(*Pump States*)
IF (iq_stPtm.i_xFault) THEN
        iq_stPtm.eState := pumpFAULT;
        iq_stPtm.xRunSW:=FALSE;
        q_RunDO:=FALSE;
ELSIF (iq_stPtm.q_RunDO) AND (iq_stPtm.i_xAtSpd) THEN
        iq_stPtm.eState := pumpRUNNING;
ELSIF (iq_stPtm.q_RunDO) AND NOT (iq_stPtm.i_xAtSpd) THEN
        iq_stPtm.eState := pumpSTARTING;
ELSIF NOT (iq_stPtm.q_RunDO) THEN
        iq_stPtm.eState := pumpSTOPPED;
ELSE
    iq_stPtm.eState := pumpFAULT;
END_IF;


(*I/O soft mapping*)
ACT_IO();
// Log States and triggers
This^.ACT_Logger();
(*Load or save the persistent variables*)
ACT_Persistent();

ACTION ACT_IO:
(*Inputs*)
iq_stPtm.i_xAtSpd := i_xAtSpd;
iq_stPtm.i_xNCError := i_xFaultNC;
iq_stPtm.i_xFault := NOT i_xFaultNC;



(*Outputs*)
iq_stPtm.q_RunDO := q_RunDO;
END_ACTION

ACTION ACT_Logger:
//STATE Logger
// ILK logger
IF NOT i_xExtIlkOK AND ePrevState = pumpRUNNING THEN
         fbLogger(sMsg:='Lost external interlock while pump was running.', eSevr:=TcEventSeverity.Critical);
END_IF


IF ePrevState <> iq_stPTM.eState THEN
      CASE iq_stPTM.eState OF
        pumpFAULT:
            fbLogger(sMsg:='Pump Fault.', eSevr:=TcEventSeverity.Critical);
          pumpSTOPPED:
            fbLogger(sMsg:='Pump stopped.', eSevr:=TcEventSeverity.Critical);
        pumpSTARTING:
            fbLogger(sMsg:='Pump starting.', eSevr:=TcEventSeverity.Info);
        pumpRUNNING:
            fbLogger(sMsg:='Pump running.', eSevr:=TcEventSeverity.Info);
      END_CASE
      ePrevState := iq_stPTM.eState;
  END_IF

// Log Action
tAction(CLK:=  iq_stPTM.q_RunDO);
IF tAction.Q THEN fbLogger(sMsg:='Pump commanded to start', eSevr:=TcEventSeverity.Info); END_IF


// Log FAULT
tFault(CLK:= NOT iq_stPTM.i_xFault);
IF tFault.Q THEN fbLogger(sMsg:='Pump Lost Alarm OK bit', eSevr:=TcEventSeverity.Critical); END_IF
END_ACTION

ACTION ACT_Persistent:
(*On first PLC pass, load the persistent value into the structrue variable*)
IF (SUPER^.bRestorePersistentData) THEN
    SUPER^.bRestorePersistentData	:= FALSE;
    IF (rBackingPressureSP <> 0) THEN
        iq_stPTM.rBackingPressureSP := rBackingPressureSP;
    END_IF;
    IF (rInletPressureSP <> 0) THEN
        iq_stPTM.rInletPressureSP := rInletPressureSP;
    END_IF;
END_IF
(*Check if a new value has been written in the structure variable copy it to the persistent variable*)
IF NOT (iq_stPTM.rBackingPressureSP = rBackingPressureSP) THEN
    rBackingPressureSP:= iq_stPTM.rBackingPressureSP;
END_IF;

IF NOT (iq_stPTM.rInletPressureSP = rInletPressureSP) THEN
    rInletPressureSP := iq_stPTM.rInletPressureSP;
END_IF;
END_ACTION

METHOD PUBLIC M_Run : BOOL
VAR_INPUT
    run:bool; // set to true to run, false to stop;
END_VAR

this^.iq_stPtm.xRunSW := run;
END_METHOD

METHOD PUBLIC M_Serial_IO : BOOL
VAR_INPUT
    i_st_TD20_RBK			: ST_TD20Status;
END_VAR

(* This function block is used to map the IO points from the Oerlikon structures
to the generic turbo structures *)

(* Readbacks *)
iq_stPTM.i_xAccel := i_st_TD20_RBK.wStatusWord.4;
iq_stPTM.i_xDecel := i_st_TD20_RBK.wStatusWord.5;
//iq_stPTM.i_xAtSpd := i_st_TD20_RBK.wStatusWord.10;
iq_stPTM.i_xRemote := i_st_TD20_RBK.wStatusWord.15; (* Remote control enabled *)
iq_stPTM.i_diCurSpd := WORD_TO_DINT(i_st_TD20_RBK.wFrequency_P3);
iq_stPTM.i_rCurrentMon := WORD_TO_INT(i_st_TD20_RBK.wMotorCurrent_P5)*0.1; (*Current in units 0.1 A, TD20 manual page 23*)
iq_stPTM.i_diPwr := LREAL_TO_DINT(WORD_TO_DINT(i_st_TD20_RBK.wMotorCurrent_P5 * i_st_TD20_RBK.wVoltage_P4)*0.01); (*Current in units 0.1 A and voltage in units 0.1V, TD20 manual page 23*)
iq_stPTM.i_diElecTemp := WORD_TO_DINT(i_st_TD20_RBK.wConverterTemp_P11);
iq_stPTM.i_rTempMon := WORD_TO_INT(i_st_TD20_RBK.wPumpTemp_P127);

(* Faults and warnings *)
//iq_stPTM.i_xFault := i_st_TD20_RBK.wStatusWord.3;
iq_stPTM.i_xTempFault := i_st_TD20_RBK.wStatusWord.7; (* specified as a temperature warning but it could be a fault *)
iq_stPTM.i_xWarn := i_st_TD20_RBK.wStatusWord.14; (* warning summary bit *)
END_METHOD

METHOD PUBLIC M_SetBackingSP
VAR_INPUT
    i_fBackingPressureSP : REAL;
END_VAR
iq_stPtm.rBackingPressureSP := i_fBackingPressureSP;
END_METHOD

METHOD PUBLIC M_SetForelineSP
VAR_INPUT
    i_fForelinePressureSP : REAL;
END_VAR
iq_stPtm.rForelineSP := i_fForelinePressureSP;
END_METHOD

END_FUNCTION_BLOCK

// ---- POUs/Functions/Pumps/FB_PTM_TwisTorr.TcPOU
(* This function block does basic controls FOR the Agilent TwisTorr 304 FS with on board Controller.
 Turns off pump in the event of errors/ warnings. Provides interlocking interface.*)
FUNCTION_BLOCK FB_PTM_TwisTorr EXTENDS FB_Pump
VAR_INPUT
    i_xExtILKOk : BOOL; // Connect to external interlock logic, TRUE if not used.
END_VAR
VAR_OUTPUT
    {attribute 'pytmc' := ' pv: '}
    iq_stPtm	:	ST_PTM;
END_VAR
VAR
    xRunOk	:	BOOL;
    (*IO*)
    i_xAtSpd AT%I*: BOOL; // Normaml operation when true
    i_xFault AT%I*: BOOL; // Error // this open collector output signal is ON when a system fault condition is detected
    q_RunDO AT%Q*: BOOL; // Start/Stop
END_VAR


(* Interlock Sum *)
iq_stPtm.xExtRunOk:= i_xExtILKOk;
xRunOk := iq_stPtm.xExtRunOk AND NOT iq_stPtm.i_xFault;

(* Basic pump supervisory section *)
IF xRunOk THEN
    iq_stPtm.q_RunDO := iq_stPTM.xRunSW;
ELSE
    iq_stPtm.xRunSW:=FALSE;
    iq_stPtm.q_RunDO:=FALSE;
END_IF

(*Pump STATE*)
IF iq_stPtm.i_xFault THEN
    iq_stPtm.eState := pumpFAULT;
ELSIF NOT iq_stPtm.q_RunDO AND NOT iq_stPTM.i_xFault THEN
    iq_stPtm.eState := pumpSTOPPED;
ELSIF NOT iq_stPtm.i_xAtSpd  AND iq_stPtm.q_RunDO THEN
    iq_stPtm.eState := pumpSTARTING;
ELSIF iq_stPtm.i_xAtSpd AND iq_stPtm.q_RunDO THEN
    iq_stPtm.eState := pumpRUNNING;
ELSE
    iq_stPtm.eState := pumpFAULT;
END_IF

(*I/O soft mapping*)
ACT_IO();
(*Log States and triggers*)
ACT_Logger();
(*Load or save the persistent variables*)
ACT_Persistent();

ACTION ACT_IO:
(*Inputs*)
iq_stPtm.i_xAtSpd := i_xAtSpd;
iq_stPtm.i_xFault := i_xFault;


(*Outputs*)
q_RunDO := iq_stPtm.q_RunDO;
END_ACTION

ACTION ACT_Logger:
//STATE Logger
// ILK logger
IF NOT i_xExtIlkOK AND ePrevState = pumpRUNNING THEN
         fbLogger(sMsg:='Lost external interlock while pump was running.', eSevr:=TcEventSeverity.Critical);
END_IF


IF ePrevState <> iq_stPTM.eState THEN
      CASE iq_stPTM.eState OF
        pumpFAULT:
            fbLogger(sMsg:='Pump Fault.', eSevr:=TcEventSeverity.Critical);
          pumpSTOPPED:
            fbLogger(sMsg:='Pump stopped.', eSevr:=TcEventSeverity.Critical);
        pumpSTARTING:
            fbLogger(sMsg:='Pump starting.', eSevr:=TcEventSeverity.Info);
        pumpRUNNING:
            fbLogger(sMsg:='Pump running.', eSevr:=TcEventSeverity.Info);
      END_CASE
      ePrevState := iq_stPTM.eState;
  END_IF

// Log Action
tAction(CLK:=  iq_stPTM.q_RunDO);
IF tAction.Q THEN fbLogger(sMsg:='Pump commanded to start', eSevr:=TcEventSeverity.Info); END_IF


// Log FAULT
tFault(CLK:= NOT iq_stPTM.i_xFault);
IF tFault.Q THEN fbLogger(sMsg:='Pump Lost Alarm OK bit', eSevr:=TcEventSeverity.Critical); END_IF
END_ACTION

ACTION ACT_Persistent:
(*On first PLC pass, load the persistent value into the structrue variable*)
IF (SUPER^.bRestorePersistentData) THEN
    SUPER^.bRestorePersistentData	:= FALSE;
    IF (rBackingPressureSP <> 0) THEN
        iq_stPTM.rBackingPressureSP := rBackingPressureSP;
    END_IF;
    IF (rInletPressureSP <> 0) THEN
        iq_stPTM.rInletPressureSP := rInletPressureSP;
    END_IF;
END_IF
(*Check if a new value has been written in the structure variable copy it to the persistent variable*)
IF NOT (iq_stPTM.rBackingPressureSP = rBackingPressureSP) THEN
    rBackingPressureSP:= iq_stPTM.rBackingPressureSP;
END_IF;

IF NOT (iq_stPTM.rInletPressureSP = rInletPressureSP) THEN
    rInletPressureSP := iq_stPTM.rInletPressureSP;
END_IF;
END_ACTION

METHOD PUBLIC M_Run : BOOL
VAR_INPUT
    run:bool; // set to true to run, false to stop;
END_VAR

this^.iq_stPtm.xRunSW := run;
END_METHOD

END_FUNCTION_BLOCK

// ---- POUs/Functions/Pumps/FB_ScrollPump.TcPOU
(* This Function block provides basic  control for Scroll Pumps *)
(* Turn on scroll pump if the Turbo Vent Valve is closed. *)
(* Cannot turn off scroll pump if turb is running. delay scroll off 150s.*)

FUNCTION_BLOCK FB_ScrollPump
VAR_IN_OUT

END_VAR
VAR_OUTPUT
    {attribute 'pytmc' := '
    pv:
    '}
    iq_stPFO	:	ST_RoughPump;
END_VAR
VAR_INPUT
    TurboIsON : BOOL;
    xExtIlk : BOOL;
END_VAR
VAR
    Tmr_TOF : TOF;
    tTimerDuration : Time:= T#150S;
    //Previous_RunSW : BOOL;
    // Digital Output to be linked
    q_xRunDo AT%Q*	:   BOOL;
END_VAR

//Turn on scroll pump if the Turbo Vent Valve is closed. So you are not just
// pumping air and accomplishing nothing

// cannot turn off scroll pump if turb is running. delay scroll off 150s.
iq_stPFO.xIlkOK := xExtIlk;// and NOT Tmr_TOF.Q;

Tmr_TOF(IN:=TurboIsON, PT := tTimerDuration);

IF iq_stPFO.xIlkOK THEN
    iq_stPFO.q_xRunDo := (Tmr_TOF.Q OR iq_stPFO.pv_xRunSW);
ELSE
    iq_stPFO.q_xRunDo := FALSE;
END_IF

iq_stPFO.pv_xRunSW := iq_stPFO.q_xRunDo;

(*State evaluation*)
IF NOT iq_stPFO.q_xRunDo THEN
    iq_stPFO.eState := pumpSTOPPED;
ELSE
    iq_stPFO.eState := pumpRUNNING;
END_IF

(*soft io Mapping*)
IO();

ACTION IO:
q_xRunDo:= iq_stPFO.q_xRunDo;
END_ACTION

METHOD PUBLIC M_Run : BOOL
VAR_INPUT
    run:bool; // set to true to run, false to stop;
END_VAR

this^.iq_stPFO.pv_xRunSW := run;
END_METHOD

END_FUNCTION_BLOCK

// ---- POUs/Functions/Pumps/functions/FB_TurboExtLogic.TcPOU
(*deprecated*)
FUNCTION_BLOCK FB_TurboExtLogic
VAR_IN_OUT
    Turbo		:	ST_AgilentPTM;
END_VAR
VAR_INPUT
    BackingGauge:	ST_VG;
    InletGauge	:	ST_VG;
    VentValve	:	ST_VCC_NO;
    ScrollPump	:	ST_RoughPump;
END_VAR
VAR_OUTPUT
END_VAR
VAR
END_VAR

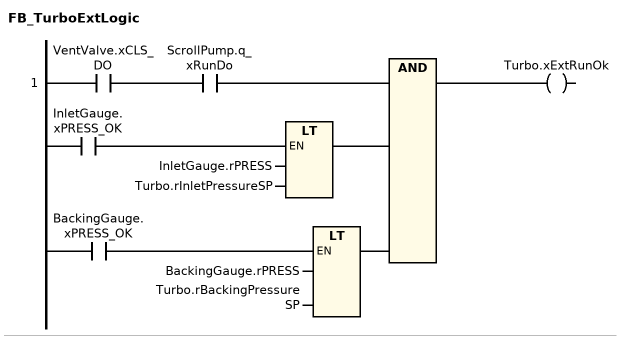
// NETWORK 1
Turbo.xExtRunOk := (VentValve.xCLS_DO AND ScrollPump.q_xRunDo) AND (InletGauge.xPRESS_OK AND InletGauge.rPRESS < Turbo.rInletPressureSP) AND (BackingGauge.xPRESS_OK AND BackingGauge.rPRESS < Turbo.rBackingPressureSP);

END_FUNCTION_BLOCK

// ---- POUs/Functions/Pumps/functions/F_TurboExtILK_NO.TcPOU
(* This function Block interfaces with a NO turbo valve*)
(* Mainly used in the FEE HXR GATT*)
FUNCTION F_TurboExtILK_NO : BOOL
VAR_INPUT
    Turbo		:	ST_PTM;
    BackingGauge:	ST_VG;
    InletGauge	:	ST_VG;
    VentValve	:	ST_VCC_NO; //NO type turbo valve
    ScrollPump	:	ST_RoughPump;
END_VAR

VAR
END_VAR

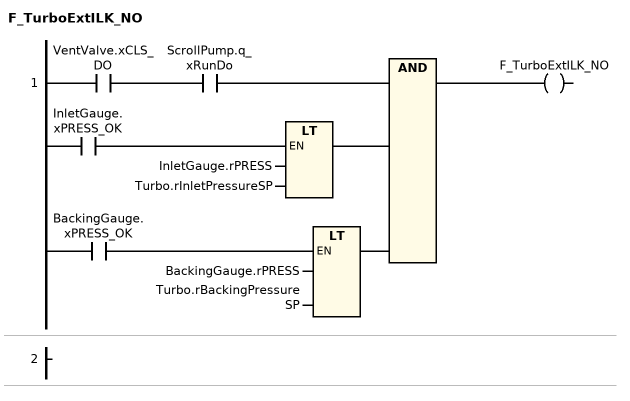
// NETWORK 1
F_TurboExtILK_NO := (VentValve.xCLS_DO AND ScrollPump.q_xRunDo) AND (InletGauge.xPRESS_OK AND InletGauge.rPRESS < Turbo.rInletPressureSP) AND (BackingGauge.xPRESS_OK AND BackingGauge.rPRESS < Turbo.rBackingPressureSP);

// NETWORK 2

END_FUNCTION

// ---- POUs/Functions/Pumps/functions/F_TurboExtILKLogic.TcPOU

(* This function evaluates the Turbo ILK logic*)
(* The Turbo shall not Run if the vent valve is open*)
(* The function also switches off the Turbo if the Inlet pressure or the backing Pressure*)
(* are higher than the configured set point*)
FUNCTION F_TurboExtILKLogic : BOOL
VAR_INPUT
    Turbo		:	ST_PTM;
    BackingGauge:	ST_VG;
    InletGauge	:	ST_VG;
    VentValve	:	ST_VVC;
    ScrollPump	:	ST_RoughPump;
END_VAR

VAR
END_VAR

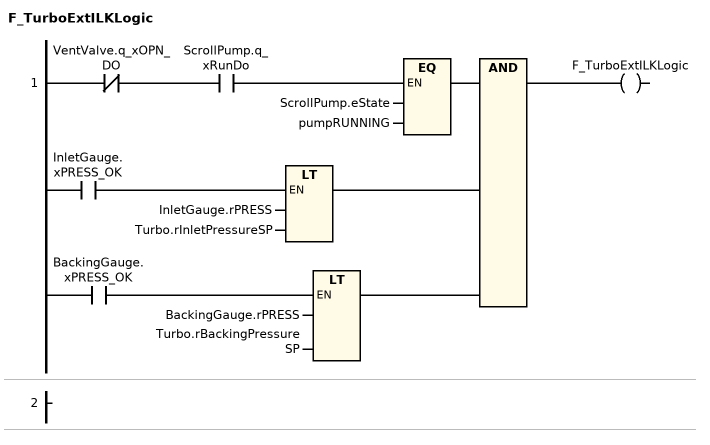
// NETWORK 1
F_TurboExtILKLogic := (NOT VentValve.q_xOPN_DO AND ScrollPump.q_xRunDo AND ScrollPump.eState = pumpRUNNING) AND (InletGauge.xPRESS_OK AND InletGauge.rPRESS < Turbo.rInletPressureSP) AND (BackingGauge.xPRESS_OK AND BackingGauge.rPRESS < Turbo.rBackingPressureSP);

// NETWORK 2

END_FUNCTION

// ---- POUs/Functions/Pumps/functions/F_TurboExtILKLogic_2.TcPOU

(* This function evaluates the Turbo ILK logic*)
(* The function switches off the Turbo if the Inlet pressure or the backing Pressure*)
(* are higher than the configured set point*)
FUNCTION F_TurboExtILKLogic_2 : BOOL
VAR_INPUT
    Turbo		:	ST_PTM;
    BackingGauge:	ST_VG;
    InletGauge	:	ST_VG;
    ScrollPump	:	ST_RoughPump;
END_VAR
VAR
END_VAR

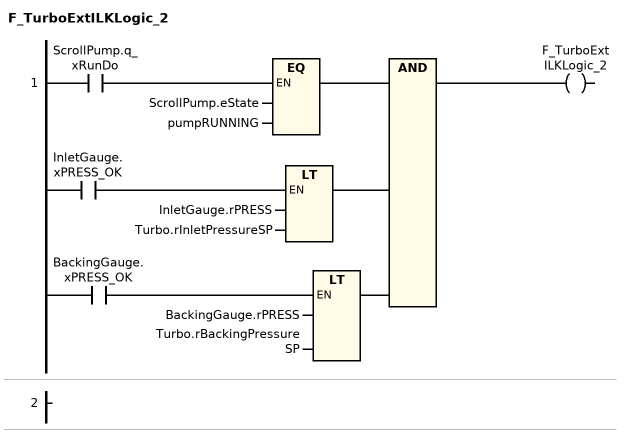
// NETWORK 1
F_TurboExtILKLogic_2 := (ScrollPump.q_xRunDo AND ScrollPump.eState = pumpRUNNING) AND (InletGauge.xPRESS_OK AND InletGauge.rPRESS < Turbo.rInletPressureSP) AND (BackingGauge.xPRESS_OK AND BackingGauge.rPRESS < Turbo.rBackingPressureSP);

// NETWORK 2

END_FUNCTION

// ---- POUs/Functions/Pumps/functions/F_TurboExtILK_NO_1.TcPOU
(* This function Block interfaces with a NO turbo valve*)
(* Mainly used in the FEE HXR GATT*)
FUNCTION F_TurboExtILK_NO_1 : BOOL
VAR_INPUT
    Turbo		:	ST_PTM;
    BackingGauge:	ST_VG;
    InletGauge	:	ST_VG;
    VentValve	:	ST_VCC_NO; //NO type turbo valve
    ScrollPump	:	ST_RoughPump;
END_VAR

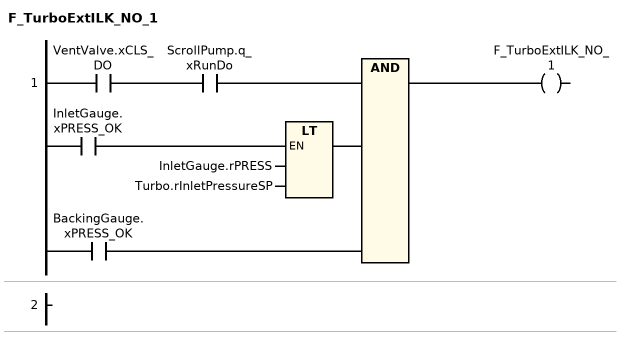
// NETWORK 1
F_TurboExtILK_NO_1 := (VentValve.xCLS_DO AND ScrollPump.q_xRunDo) AND (InletGauge.xPRESS_OK AND InletGauge.rPRESS < Turbo.rInletPressureSP) AND BackingGauge.xPRESS_OK;

// NETWORK 2

END_FUNCTION

// ---- POUs/Functions/Pumps/Interfaces/FB_PIP_Interface_In.TcPOU
(* This function block is created for interface devices between different PLC*)
(* Not all the Variables in the original structure is required, just few signals *)
(* They have to be linked to the custom created variables on the EL6692/5 primary side*)
FUNCTION_BLOCK FB_PIP_Interface_In
VAR_INPUT
END_VAR
VAR_OUTPUT
    VG : ST_VG;
END_VAR
VAR
    i_rPRESS AT%I*: REAL;  //This is the human-readable pressure
    i_xAT_VAC AT%I*: BOOL;
    i_xPRESS_OK AT%I*: BOOL;
    i_xIs_Connected AT%I*: BOOL;
END_VAR

(* This function block is created for interface devices between different PLC*)
(* Not all the Variables in the original structure is required, just few signals *)
(* They have to be linked to the custom created variables on the EL6692/5 primary side*)

VG.rPRESS := i_rPRESS;
VG.xAT_VAC := i_xAT_VAC;
VG.xPRESS_OK := i_xPRESS_OK;


IF NOT(i_xIs_Connected) THEN
    i_xPRESS_OK := FALSE;
END_IF

END_FUNCTION_BLOCK

// ---- POUs/Functions/Pumps/Interfaces/FB_PIP_Interface_Out.TcPOU
(* This function block is created for interface devices between different PLC*)
(* Not all the Variables in the original structure is required, just few signals *)
(* They have to be linked to the custom created variables on the EL6692/5 primary side*)
FUNCTION_BLOCK FB_PIP_Interface_Out
VAR_INPUT
    VG : ST_VG;
END_VAR
VAR_OUTPUT
END_VAR
VAR
    i_rPRESS AT%Q*: REAL;
    i_xAT_VAC AT%Q*: BOOL;
    i_xPRESS_OK AT%Q*: BOOL;
END_VAR

(* This function block is created for interface devices between different PLC*)
(* Not all the Variables in the original structure is required, just few signals *)
(* They have to be linked to the custom created variables on the EL6692/5 primary side*)

i_rPRESS:=VG.rPRESS;
i_xAT_VAC:= VG.xAT_VAC;
i_xPRESS_OK:=VG.xPRESS_OK;

END_FUNCTION_BLOCK

// ---- POUs/Functions/Pumps/Interfaces/FB_TPIP_ADS.TcPOU
(* This function block is created for interface devices between different PLC*)
(* Not all the Variables in the original structure is required, just few signals *)
(* The variable values are read via ADS using the symbol name*)
FUNCTION_BLOCK FB_TPIP_ADS Extends FB_ADS
VAR_INPUT
    sNetId : String; //NetID of the Destination PLC controller
    nPort : uint; // port number
    sVarName : string;// the variable name of the declared pip/pin function block.
    iWatchdog:UDINT;//The watchdog variable name written to by the remote plc
END_VAR
VAR_OUTPUT
    {attribute 'pytmc' := 'pv:'}
    IG : ST_VG;
    bError: BOOL;
END_VAR
VAR
    fb_CheckWatchdog: FB_CheckWatchdog;
    fb_Read_VG: FB_ReadAdsSymByName;
    ftReset: F_TRIG;
    xFirstPass: BOOL:= true;

END_VAR


ftReset(CLK:= fb_Read_VG.bBusy OR xFirstPass);
xFirstPass := false;
(*calling ADS read function*)

fb_Read_VG(
    bRead:=ftReset.Q ,
    sNetId:= sNetId,
    nPort:= nPort,
    sVarName:= CONCAT(sVarName,'.q_IG'),
    nDestAddr:= ADR(IG),
    nLen:= SIZEOF(IG),
    tTimeout:= ,
    eComMode:=eAdsComModeFastCom ,
    bBusy=> ,
    bError=> ,
    nErrorId=> );


(*Error*)
fb_CheckWatchdog(
    bEnable:= TRUE,
    tWatchdogTime:= T#900ms,
    nCnt:= iWatchdog ,
    bWatchdog=> ,
    nLastCnt=> );

bError:= fb_Read_VG.bError OR fb_CheckWatchdog.bWatchdog;
tErrorPresent(CLK:=bError);

IF (fb_Read_VG.bError OR fb_CheckWatchdog.bWatchdog) THEN
IG.xPRESS_OK := FALSE;
END_IF;

(*Logger*)
ACT_Logger();

ACTION ACT_Logger:
IF tErrorPresent.Q THEN
 IF(fb_Read_VG.bError) THEN fbLogger(sMsg:='ADS Read Error', eSevr:=TcEventSeverity.Critical); END_IF;
 IF(fb_CheckWatchdog.bWatchdog) THEN fbLogger(sMsg:='ADS Watchdog Error', eSevr:=TcEventSeverity.Critical); END_IF;
END_IF
END_ACTION

END_FUNCTION_BLOCK

// ---- POUs/Functions/Valves/FB_Kashiyama_VRC.TcPOU
(* Main Kashiyama gate valve permit to be open when:
        1. pump is NORMAL operating status, and
        2. chamber pressure is below HighSP or pump is at LowSpeed state.
    it will close if chamber pressure is below than lowSP for 180s.
*)
FUNCTION_BLOCK FB_Kashiyama_VRC
VAR_IN_OUT

END_VAR
VAR_OUTPUT
    {attribute 'pytmc' := ' pv:'}
    q_stValve : ST_VRC;
END_VAR
VAR_INPUT
    Pump : ST_KashiyamaDryPump;//Kashyiama pump
    i_xExtILK_OK : BOOL; //Connect to Interlock logic condition(e.g F_TURBO_VRC_ILK Function), otherwise, Set to True if the valve is not interlocked
    Gauge : ST_VG;// Pressure Gauge
    i_xOverrideMode : BOOL;
END_VAR
VAR
    At_HiVac : BOOL;
    tmrTP : TP;
    tmrPT: TIME := T#180S;
    v1: BOOL;
    tonOvrd	:	TON;
    tonDelOK : TON;
    rtOK	:	R_TRIG;

    (*IO*)
    i_xOpnLS	AT%I*: BOOL;
    i_xClsLS	AT%I*: BOOL;
    q_xOPN_DO	AT%Q*: BOOL;

END_VAR

(* Main Kashiyama gate valve permit to be open when:
        1. pump is NORMAL operating status, and
        2. chamber pressure is below HighSP or pump is at LowSpeed state.
    it will close if chamber pressure is below than lowSP for 60s.
*)
(*
      For main Kayshiyama pump's gate valve:
        Pump LowSP is MU100 base pressure (20 mTorr)
        Pump HighSP is 600 Torr;
      Second Kayshiyama pump allow Gas Attenuator operating at higher pressure,
      it's gate valve is to be open when Gas Attenuator chamber pressure is above lowSP.
*)


///Check valve postion
IF NOT q_stValve.i_xClsLS AND q_stValve.i_xOpnLS THEN
    q_stValve.eState:=OPEN;
ELSIF q_stValve.i_xClsLS AND NOT q_stValve.i_xOpnLS THEN
    q_stValve.eState:=CLOSED;
ELSIF NOT q_stValve.i_xClsLS AND NOT q_stValve.i_xOpnLS THEN
    q_stValve.eState:=MOVING;
ELSE
    q_stValve.eState:=INVALID;
END_IF

//valve open interlock
q_stValve.xOPN_OK := Pump.i_xIsRun AND Pump.RdyTmr <= 0.0 AND (Gauge.rPRESS < Pump.HighSP OR Pump.q_xLspdDo) AND i_xExtILK_OK;


(* Override logic *)
(* Goal: give ability to override, but do so in a way that people won't forget it.
Solution: Override only after ten seconds of override, protect against blips,
when the valve permission goes true for more than ten seconds consistently, remove override
*)

tonDelOK(IN:=q_stValve.xOPN_OK, PT:=T#10S);
rtOK(CLK:=tonDelOK.Q);
IF rtOK.Q THEN q_stValve.pv_xOvrdOpn :=FALSE; END_IF

//Override timer
tonOvrd(IN:=q_stValve.pv_xOvrdOpn, PT:=T#10S);


(* Here's where the valve closes *)
IF NOT q_stValve.xOPN_OK AND NOT tonOvrd.Q THEN
q_stValve.pv_xOPN_SW := FALSE;
END_IF

At_HiVac := Gauge.xPRESS_OK AND Gauge.rPRESS < Pump.LowSP;
tmrTP (IN := At_HiVac AND q_stValve.q_xOPN_DO , PT := tmrPT);

IF At_HiVac AND q_stValve.q_xOPN_DO AND NOT tmrTP.Q THEN
    q_stValve.pv_xOPN_SW := FALSE ;
END_IF

(* Here's where the valve opens *)
q_stValve.q_xOPN_DO := (q_stValve.pv_xOPN_SW AND q_stValve.xOPN_OK) OR (tonOvrd.Q AND i_xOverrideMode);

(*Soft IO Mapping*)
ACT_IO();

ACTION ACT_IO:
(*inputs*)
q_stValve.i_xOpnLS := 	i_xOpnLS;
q_stValve.i_xClsLS:=	i_xClsLS;
(*outputs*)
q_xOPN_DO:= q_stValve.q_xOPN_DO;
END_ACTION

END_FUNCTION_BLOCK

// ---- POUs/Functions/Valves/FB_MKS248.TcPOU
(* MKS248 valve using MKS1249 Drive Module *)
FUNCTION_BLOCK FB_MKS248
VAR_INPUT
    i_xExtIlkOK	:	BOOL; //External Interlock, SET to TRUE if not used
    i_rReqPos	:	REAL; //Requested position
END_VAR
VAR_OUTPUT
    {attribute 'pytmc' := 'pv:'}
    iq_stVFN	:	ST_VCN; //Needle valve structure
END_VAR
VAR CONSTANT
    rOpenVoltage	:	REAL := 9.8;
    rCloseVoltage	:	REAL := 0;
END_VAR
VAR
    // Requested voltage
    rReqVoltage: REAL := 0;
    (*IO*)
    q_iRawPosition AT%Q* :INT;
END_VAR

(* MKS248 valve using MKS1249 Drive Module *)


// Interlocking
iq_stVFN.xIlkOK := i_xExtIlkOK;
(*Checking which Control mode is selected*)
IF iq_stVFN.xIlkOK THEN
    IF iq_stVFN.eValveControl = OpenValve THEN
        iq_stVFN.rReqPosition := iq_stVFN.rUpperLimit;(*Percentage*)// iq_stVCN.rUpperLimit;
    ELSIF iq_stVFN.eValveControl = CloseValve THEN
        iq_stVFN.rReqPosition := 0; (*Percentage*)
    ELSIF iq_stVFN.eValveControl = ManualControl THEN
        iq_stVFN.rReqPosition := LIMIT(0, iq_stVFN.rReqPosition, iq_stVFN.rUpperLimit);
    ELSIF iq_stVFN.eValveControl = PressureControl THEN
        iq_stVFN.rReqPosition := LIMIT(0, i_rReqPos, iq_stVFN.rUpperLimit);
    END_IF
ELSE
    iq_stVFN.rReqPosition := 0;
    iq_stVFN.eValveControl := CloseValve;
END_IF

// Requested Voltage calculation
rReqVoltage := iq_stVFN.rReqPosition * (rOpenVoltage-rCloseVoltage)/100 + rCloseVoltage;
rReqVoltage := LIMIT(rCloseVoltage, rReqVoltage, rOpenVoltage); //The requested voltage should remain within this range
//Raw position calc
iq_stVFN.q_iRawPosition := REAL_TO_INT( 32767/10 * rReqVoltage);
(*IO Mapping*)
ACT_IO();

ACTION ACT_IO:
(*outputs*)
q_iRawPosition := iq_stVFN.q_iRawPosition;
END_ACTION

METHOD PUBLIC M_SetControlMode
VAR_INPUT
    i_eValveControlMode	:	E_VCN;
END_VAR
iq_stVFN.eValveControl := i_eValveControlMode;
END_METHOD

METHOD PUBLIC M_SetReqPosition
VAR_INPUT
    i_fReqPosition : REAL;
END_VAR
iq_stVFN.rReqPosition := i_fReqPosition;
END_METHOD

END_FUNCTION_BLOCK

// ---- POUs/Functions/Valves/FB_TurbVentvalve_NO.TcPOU
(* This function block impelemets Interlock for Agilent Turbo Vent Valve Normally Open*)
FUNCTION_BLOCK FB_TurbVentvalve_NO
VAR_OUTPUT
    {attribute 'pytmc' :=' pv:'}
    q_stValve : ST_VCC_NO;
END_VAR
VAR_INPUT
    i_stPTM	: ST_AgilentPTM; //Agilent Turbo Pump
END_VAR
VAR
    tofTmr 		: 	TOF;

    (*Output*)
    q_xCLS_DO AT%Q* : BOOL;
END_VAR

(*If the turbo is on, you cannot open the valve. In order to open the valve, you have to allow the turbopump
 to have already been turned off for 2 minutes and you have to press the open button on the vent valve

If the code looks confusing please use a truth table to verify*)

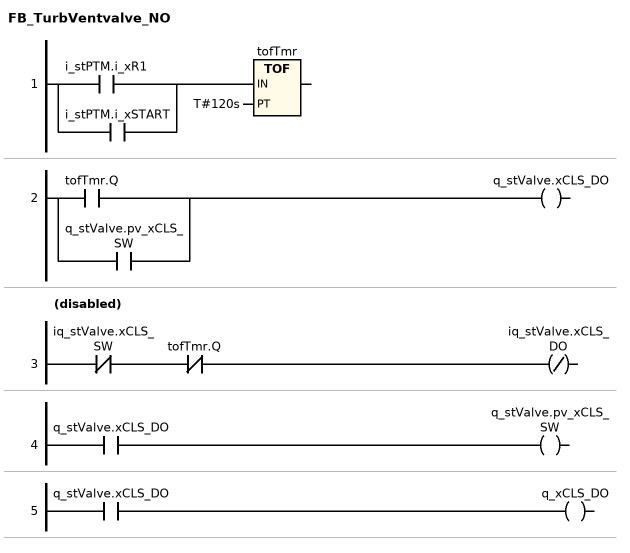
// NETWORK 1
tofTmr(IN := i_stPTM.i_xR1 OR i_stPTM.i_xSTART, PT := T#120s); // TOF

// NETWORK 2
q_stValve.xCLS_DO := tofTmr.Q OR q_stValve.pv_xCLS_SW;

// NETWORK 3 (disabled)
// iq_stValve.xCLS_DO := NOT (NOT iq_stValve.xCLS_SW AND NOT tofTmr.Q);

// NETWORK 4
q_stValve.pv_xCLS_SW := q_stValve.xCLS_DO;

// NETWORK 5
q_xCLS_DO := q_stValve.xCLS_DO;

ACTION ACT_IO:
(*outputs*)
q_xCLS_DO:= q_stValve.xCLS_DO;
END_ACTION

METHOD M_Close : BOOL
VAR_INPUT
        close:BOOL; //True to CLose, False to OPEN
END_VAR
This^.q_stValve.pv_xCLS_SW :=Close;
END_METHOD

END_FUNCTION_BLOCK

// ---- POUs/Functions/Valves/FB_Valve.TcPOU
FUNCTION_BLOCK FB_Valve
VAR_INPUT
END_VAR
VAR_OUTPUT
END_VAR
VAR
    // For logging
    fbLogger : FB_LogMessage := (eSubsystem:=E_SubSystem.VACUUM, nMinTimeViolationAcceptable:=10);
    ePrevState : E_ValvePositionState;
    tErrorPresent : R_TRIG;
    tAction : R_TRIG; // Primary action of this device (OPN_DO, etc.)
    tOverrideActivated : R_TRIG;
    // For Persistent Data
    bRestorePersistentData	:	BOOL:=TRUE;
    //fbWritePersistentData           : WritePersistentData;
END_VAR

ACTION ACT_Logger:

END_ACTION

END_FUNCTION_BLOCK

// ---- POUs/Functions/Valves/FB_VCN_VAT590.TcPOU
(* This function implements the Basic functions for the VAT590 needle valve*)
FUNCTION_BLOCK FB_VCN_VAT590 EXTENDS FB_Valve
VAR_INPUT
    bExtIlkOK : BOOL;        // External Interlock, SET to TRUE if not used
    IG : ST_VG;              // Input from a cold cathode gauge used in control loop
END_VAR
VAR_OUTPUT
    {attribute 'pytmc' := '
    pv:
    '}
    stVcnVat590	: ST_VCN_VAT590;       // Needle valve VAT590 structure
END_VAR
VAR CONSTANT
    cOpenPosition : REAL := 1E+5;      // Default position setpoint upper scale value
    cClosePosition : REAL := 0.0;      // Default position setpoint lower scale value
    cPresSPUpLim : REAL := 1E+6;       // Default pressure setpoint upper scale value
    cPresSPLowLim : REAL := 0;         // Default pressure setpoint lower scale value
    cMinPress : REAL := 1e-11;         // Default Min. pressure in Torr that can be used and requested
    cMaxPress : REAL := 1e-2;          // Default Max. pressure in Torr that can be used and requested
    cBasePress : REAL := 1E-11;        // Pressure sensor base value
    cPressRawSlope : REAL := 1E+5;     // Slope (in Units per decade) used for conversion of pressure in Torr to valve External Digital pressure sensor 1 input raw value (0-1000000)
    cPressRawBase : REAL := 1E+5;      // Valve analog output base(in Units per decade) defined for how much the curve is shifted

    cPressCtrl : ST_CoEIndSub := (nIndex := 16#2199, nSubIndex := 0); // Selected pressure controller CoE register
    cSensorDelay_AD : ST_CoEIndSub := (nIndex := 16#219A, nSubIndex := 0); // Adaptive DS controller Sensor Delay CoE register
    cRampTime_AD : ST_CoEIndSub := (nIndex := 16#219B, nSubIndex := 0); // Adaptive DS controller Ramp Time CoE register
    cRampMode_AD : ST_CoEIndSub := (nIndex := 16#219C, nSubIndex := 0); // Adaptive DS controller Ramp Mode CoE register
    cGainFactor_AD : ST_CoEIndSub := (nIndex := 16#219E, nSubIndex := 0); // Adaptive DS controller Gain factor CoE register
    cRampTime_FIX1 : ST_CoEIndSub := (nIndex := 16#21A5, nSubIndex := 0); // Fixed 1 controller Ramp Time CoE register
    cRampMode_FIX1 : ST_CoEIndSub := (nIndex := 16#21A6, nSubIndex := 0); // Fixed 1 controller Ramp Mode CoE register
    cCtrlDir_FIX1 : ST_CoEIndSub := (nIndex := 16#21A7, nSubIndex := 0); // Fixed 1 controller Control Direction CoE register
    cPGain_FIX1 : ST_CoEIndSub := (nIndex := 16#21A8, nSubIndex := 0); // Fixed 1 controller P Gain CoE register
    cIGain_FIX1 : ST_CoEIndSub := (nIndex := 16#21A9, nSubIndex := 0); // Fixed 1 controller I Gain CoE register
    cRampTime_FIX2 : ST_CoEIndSub := (nIndex := 16#21AF, nSubIndex := 0); // Fixed 2 controller Ramp Time CoE register
    cRampMode_FIX2 : ST_CoEIndSub := (nIndex := 16#21B0, nSubIndex := 0); // Fixed 2 controller Ramp Mode CoE register
    cCtrlDir_FIX2 : ST_CoEIndSub := (nIndex := 16#21B1, nSubIndex := 0); // Fixed 2 controller Control Direction CoE register
    cPGain_FIX2 : ST_CoEIndSub := (nIndex := 16#21B2, nSubIndex := 0); // Fixed 2 controller P Gain CoE register
    cIGain_FIX2 : ST_CoEIndSub := (nIndex := 16#21B3, nSubIndex := 0); // Fixed 2 controller I Gain CoE register
    cRampTime_SP : ST_CoEIndSub := (nIndex := 16#21B9, nSubIndex := 0); // Soft Pump controller Ramp Time CoE register
    cRampMode_SP : ST_CoEIndSub := (nIndex := 16#21BA, nSubIndex := 0); // Soft Pump controller Ramp Time CoE register
    cPGain_SP : ST_CoEIndSub := (nIndex := 16#21BC, nSubIndex := 0); // Soft Pump controller Ramp Time CoE register
    cPosLimitOpen : ST_CoEIndSub := (nIndex := 16#56B3, nSubIndex := 0); // General open limit. It overides the PosLimitOpenCtrl if SET lower
    cPosLimitOpenCtrl : ST_CoEIndSub := (nIndex := 16#56B4, nSubIndex := 0); // Open limit active during pressure control only
END_VAR
VAR
    fCalcPosSP : REAL := 0;
    fCalcPresSP : REAL := 0;
    fPressRaw : REAL := 0;             // Ranges 0 to 1000000 (or 0.0 to 10V) (1E-12 to 1E-2)
    eValveModeSP : E_ControlModeSP;    // Control Mode setpoint internal variable
    fReqPos : REAL;                    // Requested position internal variable
    fReqPres : REAL;                   // Requested pressure internal variable

    bRemAcsToggle : BOOL;              // Remote access control bit
    //timer for zero function
    tZeroTogg : TON := (PT := T#1S);
    //timer for remote function
    tRemAcsTogg : TON := (PT := T#500MS);
    //used for logging
    ePreviousState : E_VCN_VAT590;

    (*CoE Interface*)
    (*Link this to your VAT590 reference variables under InfoData.*)
    //Connect i_stVat590PlcDriveRef.aNetId to the VAT590 Valve InfoData^AdsAddr^netId
    //Connect i_stVat590PlcDriveRef.nSlaveAddr to the VAT590 Valve InfoData^AdsAddr^port
    i_stVat590PlcDriveRef AT %I*: ST_PlcDriveRef;
    stVat590DriveRef : ST_DriveRef;

    fbCoeRead : FB_CoERead_ByDriveRef;   // CoE Read function block
    fbCoeWrite : FB_CoEWrite_ByDriveRef; // CoE Write function block

    stCoeParamsInternal : ST_VAT590_COE;   // Internal storage of CoE parameters
    nCaseReadCoe : UINT := 1;          // Iterator for going through all CoE parameters
    rtCoeReset : R_TRIG;               // Rising edge trigger for reset CoE Interface error
    ftCoeReadBusy : F_TRIG;            // Falling edge trigger for CoE read new data
    ftCoeWriteBusy : F_TRIG;           // Falling edge trigger for CoE write data
    bFirstRead : BOOL := TRUE;         // FALSE after succesfull first readout of all CoE parameters

    (*VAT590 Ethercat IO Interface*)
    // Ethercat Interface Inputs
    i_nRawPosition       AT %I* : DINT;               // Position readback from the valve
    i_nRawPressure       AT %I* : DINT;               // Pressure readback from the valve
    i_eControlMode       AT %I* : E_ControlMode;      // Valve control mode readback
    i_eFatalError        AT %I* : E_FatalErrors;      // Valve Fatal Errors readback
    i_stGenStatus        AT %I* : ST_GeneralStatus;   // Valve General Status readback
    i_stGenWarnings      AT %I* : ST_GeneralWarnings; // Valve General Warnings readback
    i_stExtnWarnings     AT %I* : ST_ExtendedWarnings;// Valve Extended Warnings readback
    // Ethercat Interface Outputs
    o_nRawPositionSP     AT %Q* : DINT;               // Position setpoint
    o_nRawPressureSP     AT %Q* : DINT;               // Pressure setpoint
    o_nRawPressure       AT %Q* : DINT;               // Raw pressure output, eliminate need for external connection of AI, ranges 0 to 1000000 (or 0.0 to 10V) (1E-12 Torr to 1E-2 Torr)
    o_eCtrlModeSP        AT %Q* : E_ControlModeSP;    // Valve control mode setpoint
    o_stGenCtrlSP        AT %Q* : ST_GeneralControlSP;// General Control setpoint
    (*Ethercat Interface Status Check*)
    (*Link this to your VAT590 WcState variable under WcState*)
    i_bValveEthCatStatus AT %I* : BOOL := TRUE;
END_VAR
VAR PERSISTENT
    fUpperLimit	: REAL;                // Max position in % that can be requested
    fPresMaxLim : REAL;                // Max pressure in Torr that can be requested
    fPresRbMaxLim : REAL;              // Max pressure in Torr read by chamber gauge, valve will close above the pressure.
END_VAR

(* Needle valve control FB
J. Govednik 2021-11-22

This FB should be used as a low level control block.

It provides:
Valve position ceiling
Interlock
CoE Interface R/W

It could be used for:
Valve position/flow linearization
*)

(*Set Coe Interface, AmsNetID, Slave address etc*)
SetCoeInterface();

(*Read from EPICS and Valve Ethercat interface*)
ReadFromInput();

(*Checking which Control mode is selected and if valve's communication is OK*)
IF stVcnVat590.bValveEthCatStatus THEN //If valve is not connected or something is wrong with EtherCAT communication PLC will set this bit to 1
    fReqPos := 0; //set req. position to 0
    eValveModeSP := E_ControlModeSP.CloseValve; //set control mode of the valve to CLOSE VALVE
    stVcnVat590.eValveControl := E_VCN_VAT590.CloseValve; //EPICS command hold in CloseValve state
    stVcnVat590.stValveStatus.eControlMode := E_ControlMode.FatalError; //override the readback from the valve because when valve is disconnected the value remains
    stVcnVat590.nRawPosition := 0; //override the readback from the valve because when valve is disconnected the value remains
    stVcnVat590.nRawPressure := 0; //override the readback from the valve because when valve is disconnected the value remains
ELSIF bExtIlkOK THEN
    CASE stVcnVat590.eValveControl OF
        E_VCN_VAT590.OpenValve:
            eValveModeSP := E_ControlModeSP.OpenValve;
        E_VCN_VAT590.CloseValve:
            eValveModeSP := E_ControlModeSP.CloseValve;
        E_VCN_VAT590.ManualControl:
            IF IG.xPRESS_OK AND IG.rPRESS <= fPresRbMaxLim THEN
                eValveModeSP := E_ControlModeSP.ManualControl;
            ELSE
                eValveModeSP := E_ControlModeSP.CloseValve; // Close valve if something is wrong with the gauge
                stVcnVat590.eValveControl := E_VCN_VAT590.CloseValve;
            END_IF
        E_VCN_VAT590.PressureControl:
            IF IG.xPRESS_OK AND IG.rPRESS <= fPresRbMaxLim THEN
                eValveModeSP := E_ControlModeSP.PressureControl;
            ELSE
                eValveModeSP := E_ControlModeSP.CloseValve; // Close valve if something is wrong with the gauge
                stVcnVat590.eValveControl := E_VCN_VAT590.CloseValve;
            END_IF
        E_VCN_VAT590.HoldValve:
            IF stVcnVat590.stValveStatus.eControlMode = E_ControlMode.ManualControl OR
                stVcnVat590.stValveStatus.eControlMode = E_ControlMode.PressureControl THEN
                eValveModeSP := E_ControlModeSP.HoldValve;
            END_IF
    END_CASE
ELSE
    fReqPos := 0;
    eValveModeSP := E_ControlModeSP.CloseValve;
    stVcnVat590.eValveControl := E_VCN_VAT590.CloseValve;
END_IF

(*Position SP calculation*)
fReqPos := LIMIT(0, fReqPos, fUpperLimit);
fCalcPosSP := fReqPos * (cOpenPosition-cClosePosition)/100 + cClosePosition;
fCalcPosSP := LIMIT(cClosePosition, fCalcPosSP, cOpenPosition); //The requested position SP should remain within this range

(*Pressure SP calculation*)
//Limit the input from EPICS between upper and lower limit defined for seleceted pressure sensor
fReqPres := LIMIT(cMinPress, fReqPres, fPresMaxLim);
//Calcuate pressure setpoint
fCalcPresSP := cPressRawSlope * LOG(fReqPres/cBasePress) + cPressRawBase;
fCalcPresSP := LIMIT(cPresSPLowLim, fCalcPresSP, cPresSPUpLim); //The requested pressure SP should remain within this range

(*Calculated Pressure SP, Pressure readback and PressureRaw output value are 0 if Pressure sensor is not working*)
//Calculate PressureRaw value linked to the Valve's External Digital pressure sensor 1 input
//Pressure information from IG input is linked to stVcnVat590.fPressure
IF IG.xPRESS_OK THEN
    stVcnVat590.fPressure := IG.rPRESS;
    fPressRaw := cPressRawSlope * LOG(IG.rPRESS/cBasePress) + cPressRawBase;
ELSE
    fCalcPresSP := 0;
    stVcnVat590.fPressure := 0;
    fPressRaw := 0;
END_IF

(*Zero function*)
IF stVcnVat590.stValveStatus.bZeroDisabled OR tZeroTogg.Q THEN
    stVcnVat590.bZero := FALSE;
END_IF
tZeroTogg.IN := stVcnVat590.bZero;
tZeroTogg();

(*Set Remote Access*)
IF stVcnVat590.stValveStatus.eRemoteStatus <> stVcnVat590.eRemoteControl THEN
    tRemAcsTogg.IN := TRUE;
    IF tRemAcsTogg.Q THEN
        bRemAcsToggle := NOT bRemAcsToggle;
        tRemAcsTogg.IN := FALSE;
    END_IF
END_IF
tRemAcsTogg();

(*Reset Coe Interface error*)
rtCoeReset(CLK := stVcnVat590.bResetCoeError);
IF rtCoeReset.Q THEN
    stVcnVat590.bResetCoeError := FALSE;
END_IF

(*Write CoE Parameters*)
WriteCoeParameters();

(*Read CoE Parameters*)
ReadCoeParameters();

(*Write to EPICS and Valve Ethercat interface*)
WriteToOutput();

(*Load or save the persistent variables*)
LoadPersistentData();

(*Logging*)
Logger();

ACTION LoadPersistentData:
(*On first PLC pass, load the persistent value into the structrue variable*)
IF (bRestorePersistentData) THEN
    bRestorePersistentData	:= FALSE;
    IF (fUpperLimit <> 0) THEN
        stVcnVat590.fPosSetLimit := fUpperLimit;
    END_IF;
    IF (fPresMaxLim <> 0) THEN
        stVcnVat590.fPresSetLimit := fPresMaxLim;
    END_IF;
    IF (fPresRbMaxLim <> 0) THEN
        stVcnVat590.fPresRdbkLimit := fPresRbMaxLim;
    END_IF;
END_IF
END_ACTION

ACTION Logger:
// ILK logger
IF NOT (stVcnVat590.bIlkOK ) AND NOT(ePreviousState = E_VCN_VAT590.CloseValve) THEN
         fbLogger(sMsg:='Lost interlock ok bit while valve was open.', eSevr:=TcEventSeverity.Critical);
END_IF


//Control STATE Logger
IF ePreviousState <> stVcnVat590.eValveControl THEN
      CASE stVcnVat590.eValveControl OF
        E_VCN_VAT590.ManualControl:
            fbLogger(sMsg:='Valve in manual control mode.', eSevr:=TcEventSeverity.Warning);
        E_VCN_VAT590.HoldValve:
            fbLogger(sMsg:='Valve in hold control mode.', eSevr:=TcEventSeverity.Warning);
        E_VCN_VAT590.OpenValve:
            fbLogger(sMsg:='Valve Open.', eSevr:=TcEventSeverity.Info);
        E_VCN_VAT590.PressureControl:
            fbLogger(sMsg:='Valve in pressure control mode.', eSevr:=TcEventSeverity.Info);
        E_VCN_VAT590.CloseValve:
            fbLogger(sMsg:='Valve closed.', eSevr:=TcEventSeverity.Info);
      END_CASE
      ePreviousState := stVcnVat590.eValveControl;
  END_IF


// Log valve open
tAction(CLK:= (stVcnVat590.eValveControl = E_VCN_VAT590.OpenValve) );
IF tAction.Q THEN fbLogger(sMsg:='Valve commanded to fully open', eSevr:=TcEventSeverity.Info); END_IF
END_ACTION

ACTION ReadCoeParameters:
CASE nCaseReadCoe OF
    0:
        stVcnVat590.bCoeError := TRUE;
        IF rtCoeReset.Q THEN
            nCaseReadCoe := 1;
            stVcnVat590.bCoeError := FALSE;
            bFirstRead := TRUE; // Set bFirstRead after Coe interface reset
        END_IF
    1:
        fbCoeRead.nIndex := cPressCtrl.nIndex;
        fbCoeRead.nSubIndex := cPressCtrl.nSubIndex;
        fbCoeRead.pDstBuf := ADR(stVcnVat590.stCoeParameters.ePIDCtrl);
        fbCoeRead.cbBufLen := SIZEOF(stVcnVat590.stCoeParameters.ePIDCtrl);
        fbCoeRead.bExecute := TRUE;
    2:
        fbCoeRead.nIndex := cSensorDelay_AD.nIndex;
        fbCoeRead.nSubIndex := cSensorDelay_AD.nSubIndex;
        fbCoeRead.pDstBuf := ADR(stVcnVat590.stCoeParameters.fSensorDelay_AD);
        fbCoeRead.cbBufLen := SIZEOF(stVcnVat590.stCoeParameters.fSensorDelay_AD);
        fbCoeRead.bExecute := TRUE;
    3:
        fbCoeRead.nIndex := cRampTime_AD.nIndex;
        fbCoeRead.nSubIndex := cRampTime_AD.nSubIndex;
        fbCoeRead.pDstBuf := ADR(stVcnVat590.stCoeParameters.fRampTime_AD);
        fbCoeRead.cbBufLen := SIZEOF(stVcnVat590.stCoeParameters.fRampTime_AD);
        fbCoeRead.bExecute := TRUE;
    4:
        fbCoeRead.nIndex := cRampMode_AD.nIndex;
        fbCoeRead.nSubIndex := cRampMode_AD.nSubIndex;
        fbCoeRead.pDstBuf := ADR(stVcnVat590.stCoeParameters.bRampMode_AD);
        fbCoeRead.cbBufLen := SIZEOF(stVcnVat590.stCoeParameters.bRampMode_AD);
        fbCoeRead.bExecute := TRUE;
    5:
        fbCoeRead.nIndex := cGainFactor_AD.nIndex;
        fbCoeRead.nSubIndex := cGainFactor_AD.nSubIndex;
        fbCoeRead.pDstBuf := ADR(stVcnVat590.stCoeParameters.fGainFactor_AD);
        fbCoeRead.cbBufLen := SIZEOF(stVcnVat590.stCoeParameters.fGainFactor_AD);
        fbCoeRead.bExecute := TRUE;
    6:
        fbCoeRead.nIndex := cRampTime_FIX1.nIndex;
        fbCoeRead.nSubIndex := cRampTime_FIX1.nSubIndex;
        fbCoeRead.pDstBuf := ADR(stVcnVat590.stCoeParameters.fRampTime_FIX1);
        fbCoeRead.cbBufLen := SIZEOF(stVcnVat590.stCoeParameters.fRampTime_FIX1);
        fbCoeRead.bExecute := TRUE;
    7:
        fbCoeRead.nIndex := cRampMode_FIX1.nIndex;
        fbCoeRead.nSubIndex := cRampMode_FIX1.nSubIndex;
        fbCoeRead.pDstBuf := ADR(stVcnVat590.stCoeParameters.bRampMode_FIX1);
        fbCoeRead.cbBufLen := SIZEOF(stVcnVat590.stCoeParameters.bRampMode_FIX1);
        fbCoeRead.bExecute := TRUE;
    8:
        fbCoeRead.nIndex := cCtrlDir_FIX1.nIndex;
        fbCoeRead.nSubIndex := cCtrlDir_FIX1.nSubIndex;
        fbCoeRead.pDstBuf := ADR(stVcnVat590.stCoeParameters.bCtrlDir_FIX1);
        fbCoeRead.cbBufLen := SIZEOF(stVcnVat590.stCoeParameters.bCtrlDir_FIX1);
        fbCoeRead.bExecute := TRUE;
    9:
        fbCoeRead.nIndex := cPGain_FIX1.nIndex;
        fbCoeRead.nSubIndex := cPGain_FIX1.nSubIndex;
        fbCoeRead.pDstBuf := ADR(stVcnVat590.stCoeParameters.fPGain_FIX1);
        fbCoeRead.cbBufLen := SIZEOF(stVcnVat590.stCoeParameters.fPGain_FIX1);
        fbCoeRead.bExecute := TRUE;
    10:
        fbCoeRead.nIndex := cIGain_FIX1.nIndex;
        fbCoeRead.nSubIndex := cIGain_FIX1.nSubIndex;
        fbCoeRead.pDstBuf := ADR(stVcnVat590.stCoeParameters.fIGain_FIX1);
        fbCoeRead.cbBufLen := SIZEOF(stVcnVat590.stCoeParameters.fIGain_FIX1);
        fbCoeRead.bExecute := TRUE;
    11:
        fbCoeRead.nIndex := cRampTime_FIX2.nIndex;
        fbCoeRead.nSubIndex := cRampTime_FIX2.nSubIndex;
        fbCoeRead.pDstBuf := ADR(stVcnVat590.stCoeParameters.fRampTime_FIX2);
        fbCoeRead.cbBufLen := SIZEOF(stVcnVat590.stCoeParameters.fRampTime_FIX2);
        fbCoeRead.bExecute := TRUE;
    12:
        fbCoeRead.nIndex := cRampMode_FIX2.nIndex;
        fbCoeRead.nSubIndex := cRampMode_FIX2.nSubIndex;
        fbCoeRead.pDstBuf := ADR(stVcnVat590.stCoeParameters.bRampMode_FIX2);
        fbCoeRead.cbBufLen := SIZEOF(stVcnVat590.stCoeParameters.bRampMode_FIX2);
        fbCoeRead.bExecute := TRUE;
    13:
        fbCoeRead.nIndex := cCtrlDir_FIX2.nIndex;
        fbCoeRead.nSubIndex := cCtrlDir_FIX2.nSubIndex;
        fbCoeRead.pDstBuf := ADR(stVcnVat590.stCoeParameters.bCtrlDir_FIX2);
        fbCoeRead.cbBufLen := SIZEOF(stVcnVat590.stCoeParameters.bCtrlDir_FIX2);
        fbCoeRead.bExecute := TRUE;
    14:
        fbCoeRead.nIndex := cPGain_FIX2.nIndex;
        fbCoeRead.nSubIndex := cPGain_FIX2.nSubIndex;
        fbCoeRead.pDstBuf := ADR(stVcnVat590.stCoeParameters.fPGain_FIX2);
        fbCoeRead.cbBufLen := SIZEOF(stVcnVat590.stCoeParameters.fPGain_FIX2);
        fbCoeRead.bExecute := TRUE;
    15:
        fbCoeRead.nIndex := cIGain_FIX2.nIndex;
        fbCoeRead.nSubIndex := cIGain_FIX2.nSubIndex;
        fbCoeRead.pDstBuf := ADR(stVcnVat590.stCoeParameters.fIGain_FIX2);
        fbCoeRead.cbBufLen := SIZEOF(stVcnVat590.stCoeParameters.fIGain_FIX2);
        fbCoeRead.bExecute := TRUE;
    16:
        fbCoeRead.nIndex := cRampTime_SP.nIndex;
        fbCoeRead.nSubIndex := cRampTime_SP.nSubIndex;
        fbCoeRead.pDstBuf := ADR(stVcnVat590.stCoeParameters.fRampTime_SP);
        fbCoeRead.cbBufLen := SIZEOF(stVcnVat590.stCoeParameters.fRampTime_SP);
        fbCoeRead.bExecute := TRUE;
    17:
        fbCoeRead.nIndex := cRampMode_SP.nIndex;
        fbCoeRead.nSubIndex := cRampMode_SP.nSubIndex;
        fbCoeRead.pDstBuf := ADR(stVcnVat590.stCoeParameters.bRampMode_SP);
        fbCoeRead.cbBufLen := SIZEOF(stVcnVat590.stCoeParameters.bRampMode_SP);
        fbCoeRead.bExecute := TRUE;
    18:
        fbCoeRead.nIndex := cPGain_SP.nIndex;
        fbCoeRead.nSubIndex := cPGain_SP.nSubIndex;
        fbCoeRead.pDstBuf := ADR(stVcnVat590.stCoeParameters.fPGain_SP);
        fbCoeRead.cbBufLen := SIZEOF(stVcnVat590.stCoeParameters.fPGain_SP);
        fbCoeRead.bExecute := TRUE;
    19:
        fbCoeRead.nIndex := cPosLimitOpen.nIndex;
        fbCoeRead.nSubIndex := cPosLimitOpen.nSubIndex;
        fbCoeRead.pDstBuf := ADR(stVcnVat590.stCoeParameters.fPositionLimitOpen);
        fbCoeRead.cbBufLen := SIZEOF(stVcnVat590.stCoeParameters.fPositionLimitOpen);
        fbCoeRead.bExecute := TRUE;
    20:
        fbCoeRead.nIndex := cPosLimitOpenCtrl.nIndex;
        fbCoeRead.nSubIndex := cPosLimitOpenCtrl.nSubIndex;
        fbCoeRead.pDstBuf := ADR(stVcnVat590.stCoeParameters.fPositionLimitOpenControl);
        fbCoeRead.cbBufLen := SIZEOF(stVcnVat590.stCoeParameters.fPositionLimitOpenControl);
        fbCoeRead.bExecute := TRUE;
END_CASE

ftCoeReadBusy(CLK:=fbCoeRead.bBusy);
IF ftCoeReadBusy.Q THEN
    fbCoeRead.bExecute := FALSE;
    IF NOT fbCoeRead.bError THEN
        nCaseReadCoe := nCaseReadCoe + 1;
        IF nCaseReadCoe > 20 THEN
            nCaseReadCoe := 1;
            bFirstRead := FALSE; // Reset bFirstRead after successfull readout of all parameters
        END_IF
    ELSE
        nCaseReadCoe := 0; // Go to Error state
    END_IF
END_IF

fbCoeRead();
stCoeParamsInternal := stVcnVat590.stCoeParameters; //Save current values to internal structure
END_ACTION

ACTION ReadFromInput:
(*Read from EPICS*)
fUpperLimit := LIMIT(0, stVcnVat590.fPosSetLimit, 100);
fPresMaxLim := LIMIT(cMinPress, stVcnVat590.fPresSetLimit, cMaxPress);
fPresRbMaxLim := LIMIT(cMinPress, stVcnVat590.fPresRdbkLimit, cMaxPress);
fReqPos := LIMIT(0, stVcnVat590.fReqPosition, 100);
fReqPres := LIMIT(cMinPress, stVcnVat590.fReqPressure, cMaxPress);

(*Read from VAT valve*)
stVcnVat590.stValveStatus.eControlMode := i_eControlMode;
stVcnVat590.stValveStatus.eFatalErrors := i_eFatalError;
stVcnVat590.nRawPosition := i_nRawPosition;
stVcnVat590.nRawPressure := i_nRawPressure;
//Mapping General statuses
stVcnVat590.stValveStatus.bFieldBusDatavalid := i_stGenStatus.Bit0FieldBusDatavalid;
stVcnVat590.stValveStatus.bZeroExecuted := i_stGenStatus.Bit1ZeroExecuted;
stVcnVat590.stValveStatus.bPingPongRxBit := i_stGenStatus.Bit2PingPongRxBit;
stVcnVat590.stValveStatus.bPressureSimulation := i_stGenStatus.Bit3PressureSimulation;
stVcnVat590.stValveStatus.bPressureSPReached := i_stGenStatus.Bit4PressureSPReached;
stVcnVat590.stValveStatus.bWarningsActive := i_stGenStatus.Bit9WarningsActive;
//Read Remote status
stVcnVat590.stValveStatus.eRemoteStatus.0 := i_stGenStatus.Bit7AccessModeBit0;
stVcnVat590.stValveStatus.eRemoteStatus.1 := i_stGenStatus.Bit8AccessModeBit1;
//Mapping General warnings
stVcnVat590.stValveStatus.bServiceRequest := i_stGenWarnings.Bit0ServiceRequest;
stVcnVat590.stValveStatus.bPowerFailureBattery := i_stGenWarnings.Bit3PowerFailureBattery;
stVcnVat590.stValveStatus.bSensMeasUnitFault := i_stGenWarnings.Bit10SensMeasUnitFault;
//Mapping Extended warnings
stVcnVat590.stValveStatus.bRemoteControlNotPossible := i_stExtnWarnings.Bit0RemoteControlNotPossible;
stVcnVat590.stValveStatus.bControlModeSPNotAllowed := i_stExtnWarnings.Bit1ControlModeSPNotAllowed;
stVcnVat590.stValveStatus.bZeroDisabled := i_stExtnWarnings.Bit2ZeroDisabled;
stVcnVat590.stValveStatus.bPFODeactivated := i_stExtnWarnings.Bit3PFODeactivated;
stVcnVat590.stValveStatus.bPressureSPOutOfRange := i_stExtnWarnings.Bit5PressureSPOutOfRange;
stVcnVat590.stValveStatus.bPositionSPOutOfRange := i_stExtnWarnings.Bit6PositionSPOutOfRange;
stVcnVat590.stValveStatus.bCtrlSPOutOfRange := i_stExtnWarnings.Bit10CtrlSPOutOfRange;
stVcnVat590.stValveStatus.bGeneralCtrlSPOutOfRange := i_stExtnWarnings.Bit11GeneralCtrlSPOutOfRange;
stVcnVat590.stValveStatus.bProcDataSettingsNotvalid := i_stExtnWarnings.Bit12ProcDataSettingsNotvalid;
//Mapping WcState - Valve Ethercat Status
stVcnVat590.bValveEthCatStatus := i_bValveEthCatStatus;
END_ACTION

ACTION SetCoeInterface:
stVat590DriveRef.sNetId := F_CreateAmsNetId(i_stVat590PlcDriveRef.aNetId);
stVat590DriveRef.nSlaveAddr := i_stVat590PlcDriveRef.nSlaveAddr;
stVat590DriveRef.nDriveNo := i_stVat590PlcDriveRef.nDriveNo;
stVat590DriveRef.nDriveType := i_stVat590PlcDriveRef.nDriveType;
fbCoeRead.stDriveRef := stVat590DriveRef;
fbCoeWrite.stDriveRef := stVat590DriveRef;
END_ACTION

METHOD SetThrottle : BOOL
VAR_INPUT
    rUpperLimit	:	REAL;
END_VAR
stVcnVat590.fPosSetLimit := LIMIT(0, rUpperLimit, 100);
END_METHOD

METHOD ValveControl : BOOL
VAR_INPUT
    state : E_VCN_VAT590; // Set Control modes
END_VAR
stVcnVat590.eValveControl := state;
END_METHOD

ACTION WriteCoeParameters:
// User will change one parameter at a time so solution with ELSIF should work OK
IF stVcnVat590.bCoeError THEN
    IF rtCoeReset.Q THEN
        stVcnVat590.bCoeError := FALSE;
    END_IF;
ELSIF bFirstRead THEN
    ;//Wait until first readout of all CoE parameters is completed
ELSIF stVcnVat590.stCoeParameters.ePIDCtrl <> stCoeParamsInternal.ePIDCtrl THEN
    fbCoeWrite.nIndex := cPressCtrl.nIndex;
    fbCoeWrite.nSubIndex := cPressCtrl.nSubIndex;
    fbCoeWrite.pSrcBuf := ADR(stVcnVat590.stCoeParameters.ePIDCtrl);
    fbCoeWrite.cbBufLen := SIZEOF(stVcnVat590.stCoeParameters.ePIDCtrl);
    fbCoeWrite.bExecute := TRUE;
ELSIF stVcnVat590.stCoeParameters.fSensorDelay_AD <> stCoeParamsInternal.fSensorDelay_AD THEN
    fbCoeWrite.nIndex := cSensorDelay_AD.nIndex;
    fbCoeWrite.nSubIndex := cSensorDelay_AD.nSubIndex;
    fbCoeWrite.pSrcBuf := ADR(stVcnVat590.stCoeParameters.fSensorDelay_AD);
    fbCoeWrite.cbBufLen := SIZEOF(stVcnVat590.stCoeParameters.fSensorDelay_AD);
    fbCoeWrite.bExecute := TRUE;
ELSIF stVcnVat590.stCoeParameters.fRampTime_AD <> stCoeParamsInternal.fRampTime_AD THEN
    fbCoeWrite.nIndex := cRampTime_AD.nIndex;
    fbCoeWrite.nSubIndex := cRampTime_AD.nSubIndex;
    fbCoeWrite.pSrcBuf := ADR(stVcnVat590.stCoeParameters.fRampTime_AD);
    fbCoeWrite.cbBufLen := SIZEOF(stVcnVat590.stCoeParameters.fRampTime_AD);
    fbCoeWrite.bExecute := TRUE;
ELSIF stVcnVat590.stCoeParameters.bRampMode_AD <> stCoeParamsInternal.bRampMode_AD THEN
    fbCoeWrite.nIndex := cRampMode_AD.nIndex;
    fbCoeWrite.nSubIndex := cRampMode_AD.nSubIndex;
    fbCoeWrite.pSrcBuf := ADR(stVcnVat590.stCoeParameters.bRampMode_AD);
    fbCoeWrite.cbBufLen := SIZEOF(stVcnVat590.stCoeParameters.bRampMode_AD);
    fbCoeWrite.bExecute := TRUE;
ELSIF stVcnVat590.stCoeParameters.fGainFactor_AD <> stCoeParamsInternal.fGainFactor_AD THEN
    fbCoeWrite.nIndex := cGainFactor_AD.nIndex;
    fbCoeWrite.nSubIndex := cGainFactor_AD.nSubIndex;
    fbCoeWrite.pSrcBuf := ADR(stVcnVat590.stCoeParameters.fGainFactor_AD);
    fbCoeWrite.cbBufLen := SIZEOF(stVcnVat590.stCoeParameters.fGainFactor_AD);
    fbCoeWrite.bExecute := TRUE;
ELSIF stVcnVat590.stCoeParameters.fRampTime_FIX1 <> stCoeParamsInternal.fRampTime_FIX1 THEN
    fbCoeWrite.nIndex := cRampTime_FIX1.nIndex;
    fbCoeWrite.nSubIndex := cRampTime_FIX1.nSubIndex;
    fbCoeWrite.pSrcBuf := ADR(stVcnVat590.stCoeParameters.fRampTime_FIX1);
    fbCoeWrite.cbBufLen := SIZEOF(stVcnVat590.stCoeParameters.fRampTime_FIX1);
    fbCoeWrite.bExecute := TRUE;
ELSIF stVcnVat590.stCoeParameters.bRampMode_FIX1 <> stCoeParamsInternal.bRampMode_FIX1 THEN
    fbCoeWrite.nIndex := cRampMode_FIX1.nIndex;
    fbCoeWrite.nSubIndex := cRampMode_FIX1.nSubIndex;
    fbCoeWrite.pSrcBuf := ADR(stVcnVat590.stCoeParameters.bRampMode_FIX1);
    fbCoeWrite.cbBufLen := SIZEOF(stVcnVat590.stCoeParameters.bRampMode_FIX1);
    fbCoeWrite.bExecute := TRUE;
ELSIF stVcnVat590.stCoeParameters.bCtrlDir_FIX1 <> stCoeParamsInternal.bCtrlDir_FIX1 THEN
    fbCoeWrite.nIndex := cCtrlDir_FIX1.nIndex;
    fbCoeWrite.nSubIndex := cCtrlDir_FIX1.nSubIndex;
    fbCoeWrite.pSrcBuf := ADR(stVcnVat590.stCoeParameters.bCtrlDir_FIX1);
    fbCoeWrite.cbBufLen := SIZEOF(stVcnVat590.stCoeParameters.bCtrlDir_FIX1);
    fbCoeWrite.bExecute := TRUE;
ELSIF stVcnVat590.stCoeParameters.fPGain_FIX1 <> stCoeParamsInternal.fPGain_FIX1 THEN
    fbCoeWrite.nIndex := cPGain_FIX1.nIndex;
    fbCoeWrite.nSubIndex := cPGain_FIX1.nSubIndex;
    fbCoeWrite.pSrcBuf := ADR(stVcnVat590.stCoeParameters.fPGain_FIX1);
    fbCoeWrite.cbBufLen := SIZEOF(stVcnVat590.stCoeParameters.fPGain_FIX1);
    fbCoeWrite.bExecute := TRUE;
ELSIF stVcnVat590.stCoeParameters.fIGain_FIX1 <> stCoeParamsInternal.fIGain_FIX1 THEN
    fbCoeWrite.nIndex := cIGain_FIX1.nIndex;
    fbCoeWrite.nSubIndex := cIGain_FIX1.nSubIndex;
    fbCoeWrite.pSrcBuf := ADR(stVcnVat590.stCoeParameters.fIGain_FIX1);
    fbCoeWrite.cbBufLen := SIZEOF(stVcnVat590.stCoeParameters.fIGain_FIX1);
    fbCoeWrite.bExecute := TRUE;
ELSIF stVcnVat590.stCoeParameters.fRampTime_FIX2 <> stCoeParamsInternal.fRampTime_FIX2 THEN
    fbCoeWrite.nIndex := cRampTime_FIX2.nIndex;
    fbCoeWrite.nSubIndex := cRampTime_FIX2.nSubIndex;
    fbCoeWrite.pSrcBuf := ADR(stVcnVat590.stCoeParameters.fRampTime_FIX2);
    fbCoeWrite.cbBufLen := SIZEOF(stVcnVat590.stCoeParameters.fRampTime_FIX2);
    fbCoeWrite.bExecute := TRUE;
ELSIF stVcnVat590.stCoeParameters.bRampMode_FIX2 <> stCoeParamsInternal.bRampMode_FIX2 THEN
    fbCoeWrite.nIndex := cRampMode_FIX2.nIndex;
    fbCoeWrite.nSubIndex := cRampMode_FIX2.nSubIndex;
    fbCoeWrite.pSrcBuf := ADR(stVcnVat590.stCoeParameters.bRampMode_FIX2);
    fbCoeWrite.cbBufLen := SIZEOF(stVcnVat590.stCoeParameters.bRampMode_FIX2);
    fbCoeWrite.bExecute := TRUE;
ELSIF stVcnVat590.stCoeParameters.bCtrlDir_FIX2 <> stCoeParamsInternal.bCtrlDir_FIX2 THEN
    fbCoeWrite.nIndex := cCtrlDir_FIX2.nIndex;
    fbCoeWrite.nSubIndex := cCtrlDir_FIX2.nSubIndex;
    fbCoeWrite.pSrcBuf := ADR(stVcnVat590.stCoeParameters.bCtrlDir_FIX2);
    fbCoeWrite.cbBufLen := SIZEOF(stVcnVat590.stCoeParameters.bCtrlDir_FIX2);
    fbCoeWrite.bExecute := TRUE;
ELSIF stVcnVat590.stCoeParameters.fPGain_FIX2 <> stCoeParamsInternal.fPGain_FIX2 THEN
    fbCoeWrite.nIndex := cPGain_FIX2.nIndex;
    fbCoeWrite.nSubIndex := cPGain_FIX2.nSubIndex;
    fbCoeWrite.pSrcBuf := ADR(stVcnVat590.stCoeParameters.fPGain_FIX2);
    fbCoeWrite.cbBufLen := SIZEOF(stVcnVat590.stCoeParameters.fPGain_FIX2);
    fbCoeWrite.bExecute := TRUE;
ELSIF stVcnVat590.stCoeParameters.fIGain_FIX2 <> stCoeParamsInternal.fIGain_FIX2 THEN
    fbCoeWrite.nIndex := cIGain_FIX2.nIndex;
    fbCoeWrite.nSubIndex := cIGain_FIX2.nSubIndex;
    fbCoeWrite.pSrcBuf := ADR(stVcnVat590.stCoeParameters.fIGain_FIX2);
    fbCoeWrite.cbBufLen := SIZEOF(stVcnVat590.stCoeParameters.fIGain_FIX2);
    fbCoeWrite.bExecute := TRUE;
ELSIF stVcnVat590.stCoeParameters.fRampTime_SP <> stCoeParamsInternal.fRampTime_SP THEN
    fbCoeWrite.nIndex := cRampTime_SP.nIndex;
    fbCoeWrite.nSubIndex := cRampTime_SP.nSubIndex;
    fbCoeWrite.pSrcBuf := ADR(stVcnVat590.stCoeParameters.fRampTime_SP);
    fbCoeWrite.cbBufLen := SIZEOF(stVcnVat590.stCoeParameters.fRampTime_SP);
    fbCoeWrite.bExecute := TRUE;
ELSIF stVcnVat590.stCoeParameters.bRampMode_SP <> stCoeParamsInternal.bRampMode_SP THEN
    fbCoeWrite.nIndex := cRampMode_SP.nIndex;
    fbCoeWrite.nSubIndex := cRampMode_SP.nSubIndex;
    fbCoeWrite.pSrcBuf := ADR(stVcnVat590.stCoeParameters.bRampMode_SP);
    fbCoeWrite.cbBufLen := SIZEOF(stVcnVat590.stCoeParameters.bRampMode_SP);
    fbCoeWrite.bExecute := TRUE;
ELSIF stVcnVat590.stCoeParameters.fPGain_SP <> stCoeParamsInternal.fPGain_SP THEN
    fbCoeWrite.nIndex := cPGain_SP.nIndex;
    fbCoeWrite.nSubIndex := cPGain_SP.nSubIndex;
    fbCoeWrite.pSrcBuf := ADR(stVcnVat590.stCoeParameters.fPGain_SP);
    fbCoeWrite.cbBufLen := SIZEOF(stVcnVat590.stCoeParameters.fPGain_SP);
    fbCoeWrite.bExecute := TRUE;
ELSIF stVcnVat590.stCoeParameters.fPositionLimitOpen <> stCoeParamsInternal.fPositionLimitOpen THEN
    fbCoeWrite.nIndex := cPosLimitOpen.nIndex;
    fbCoeWrite.nSubIndex := cPosLimitOpen.nSubIndex;
    fbCoeWrite.pSrcBuf := ADR(stVcnVat590.stCoeParameters.fPositionLimitOpen);
    fbCoeWrite.cbBufLen := SIZEOF(stVcnVat590.stCoeParameters.fPositionLimitOpen);
    fbCoeWrite.bExecute := TRUE;
ELSIF stVcnVat590.stCoeParameters.fPositionLimitOpenControl <> stCoeParamsInternal.fPositionLimitOpenControl THEN
    fbCoeWrite.nIndex := cPosLimitOpenCtrl.nIndex;
    fbCoeWrite.nSubIndex := cPosLimitOpenCtrl.nSubIndex;
    fbCoeWrite.pSrcBuf := ADR(stVcnVat590.stCoeParameters.fPositionLimitOpenControl);
    fbCoeWrite.cbBufLen := SIZEOF(stVcnVat590.stCoeParameters.fPositionLimitOpenControl);
    fbCoeWrite.bExecute := TRUE;
END_IF

ftCoeWriteBusy(CLK:=fbCoeWrite.bBusy);
IF ftCoeWriteBusy.Q THEN
    fbCoeWrite.bExecute := FALSE;
    IF fbCoeWrite.bError THEN
        stVcnVat590.bCoeError := TRUE;
    END_IF
END_IF

fbCoeWrite();
END_ACTION

ACTION WriteToOutput:
(*Write to EPICS*)
stVcnVat590.bIlkOK := bExtIlkOK;
stVcnVat590.nPositionSP := REAL_TO_DINT(fCalcPosSP);
stVcnVat590.nPressureSP := REAL_TO_DINT(fCalcPresSP);
stVcnVat590.fReqPosition := fReqPos;
stVcnVat590.fReqPressure := fReqPres;
stVcnVat590.fPresSetLimit := fPresMaxLim;
stVcnVat590.fPosSetLimit := fUpperLimit;

(*Write to VAT valve*)
o_eCtrlModeSP := eValveModeSP;
o_nRawPositionSP := REAL_TO_DINT(fCalcPosSP);
o_nRawPressureSP := REAL_TO_DINT(fCalcPresSP);
o_nRawPressure := REAL_TO_DINT(fPressRaw);
o_stGenCtrlSP.Bit0ExecuteZero := stVcnVat590.bZero;
o_stGenCtrlSP.Bit4AccessMode := bRemAcsToggle;
END_ACTION

END_FUNCTION_BLOCK

// ---- POUs/Functions/Valves/FB_VFS.TcPOU
(* This function block implements basic functionality for Fast Shutter/Valves*)
(* Create a separate virtual PLC for the fast shutter logic, and tie/map this task to the FAST I/O portion of the ethercat bus,
 so we can scan these I/Os faster than the rest of the vacuum I/Os.
The Fast shutter was tested with PLC task Cycle Base Time 50us with cycle time 0.050ms.
*)
FUNCTION_BLOCK FB_VFS EXTENDS FB_Valve
VAR_INPUT
    i_xPMPS_OK:	BOOL	; (*External MPS interlock, Set to TRUE when no PMPS interlock is required*)
    i_xExt_OK: BOOL; (*Other External Interlock, Set to True when no external interlock is required*)
    i_sDevName : T_MaxString :=  'VGC'; // Device name for diagnostic
    i_xVeto_Enable:BOOL:= FALSE; (*Set to TRUE if there is a Veto Valve to this VFS*)
END_VAR
VAR_IN_OUT
    io_fbFFHWO    :    FB_HardwareFFOutput;
END_VAR
VAR
    xOPN_OK :BOOL;
    xERR_ExtFault :BOOL;
    xVeto: BOOL;
    // PMPS
    fbFF    :    FB_FastFault :=(
        i_DevName := 'VFS',
        i_Desc := 'Fault occurs when fast valve is not in open state',
        i_TypeCode := 16#1010);

    rDiffPressAllowed	:	REAL := 22.5; // Torr, Default value comes from Vat Valve Manual
    rDiffPress : REAL;
    set : BOOL;
    reset: BOOL;

    xFirstPass	:	BOOL := TRUE;
    //fbFSInit		:	R_TRIG;
    rtOPN_SW :	R_TRIG;

    tonDelOK : TON;
    rtOK	:	R_TRIG;
    tonOvrd	:	TON;

    tDelOK	:	TIME := T#60S;
    tOvrd	:	TIME := T#10s;
    rTrigOverrideOpen : R_TRIG;

    xClose: BOOL;
    xOpen: BOOL;
    CloseTimer: TON;
    TimDur: TIME := T#20MS;
    OpenTimer: TON;
    OpenTimDur: TIME := T#2S;

    (* Timeouts*)
    tCLSTimeOutDuration: TIME:= T#0.5S;
    tOPNTimeOutDuration: TIME:= T#10S;
    tOPNtimeout: TON;
    tCLStimeout:TON;


    (*IO*)
    i_xOpnLS	AT%I*: BOOL;
    i_xClsLS	AT%I*: BOOL;
    q_xClose_A	AT%Q*: BOOL;
    q_xClose_B	AT%Q*: BOOL;
    q_xClose_C	AT%Q*: BOOL;
    q_xOPN_DO	AT%Q*: BOOL;
    i_xTrigger	AT%I*: BOOL;

    (*VETO Devices*)
    i_xVetoValveOpenDO AT%I*: BOOL;
    i_xVetoValveClosed AT%I*: BOOL;

    // Interface
    i_xPress_OK AT%I*:BOOL; (*To be linked to the Fast sensor structure signal IG.xPRESS_OK, to make sure that the device is connected*)
    i_xOPN_SW AT%I*:BOOL;
    i_xCLS_SW AT%I*:BOOL; (*external open signal e.g epics*)
    i_xVAC_FAULT_Reset	AT%I*: BOOL;(*Valve Vacuum OK, is set to False when there is Vacuum Fault*)
    i_xOverrideMode AT%I*: BOOL; (*To be linked to global override bit. This Overrides Vacuum logic only, EPS, MPS and PMPS are still enforces*)
    i_xOverrideOpen AT%I*: BOOL;
    q_xTrigger	AT%Q*: BOOL; (*Interface*)
    q_xVFS_Open AT%Q*: BOOL; (*Interface*)
    q_xVFS_Closed AT%Q*: BOOL; (*Interface*)
    q_xVAC_FAULT_OK AT%Q*: BOOL; (*Valve Vacuum OK, is set to False when there is Vacuum Fault*)
    q_xMPS_OK	 AT%Q*:	BOOL; (*MPS Fault OK, is set when the Valve is Open and there is no trigger*)
    q_eVFS_State AT%Q*: E_VGC; (*Interface*)

END_VAR



(* Fast Shutter/Valve Function Block*)
(* M.Ghaly Feb 2019*)

(* Fast Shutters do not function as complete isolation valves, but are intended to rapidly limit conductance
between vacuum regions.  They should be installed in conjunction with isolation gate valves.  The conductance
of the fast shutter in the closed state may be sufficiently low as to create an isolated vacuum region.
Thus, at least a pirani gauge, that can measure a pressure down to 1x10-4 Torr, needs to be installed between
the shutter and the isolation gate valve.
In the case where a gauge is not installed, the neigboring gate Valves should not be opened unless the shutter
is Open.
*)
(* On first PLC pass, put valve into vented state, which implies a closed valve *)
IF xFirstPass THEN
    fbFF.i_DevName := i_sDevName;
    xFirstPass := FALSE;
END_IF


(*set Veto bit*)
IF (i_xVeto_Enable) THEN
    xVeto := (i_xVetoValveClosed AND NOT i_xVetoValveOpenDO);
    ELSE xVeto:=FALSE;
END_IF

//xVeto:= i_xVeto AND (i_xVetoValveClosed AND NOT i_xVetoValveOpenDO);
(* Input Trigger to close the Fast Shutter*)
(* Neighboring Valves Should also be triggered to Close*)
IF ((i_xTrigger) OR NOT (i_xPress_OK) OR NOT (i_xExt_OK))  AND NOT(xVeto) AND NOT (tonOvrd.Q AND i_xOverrideMode) THEN
    xClose:= TRUE;
    xOpen:= FALSE;
    q_xVAC_FAULT_OK:= FALSE;
    xERR_ExtFault := TRUE; ;
    i_xCLS_SW := TRUE;
    q_xOPN_DO := FALSE;
    //i_xOPN_SW :=FALSE;
    xOpen:=FALSE;
ELSIF (i_xCLS_SW) THEN
    xClose:= TRUE;
    xOpen:= FALSE;
    q_xVAC_FAULT_OK:= FALSE;
    i_xCLS_SW := TRUE;
    q_xOPN_DO := FALSE;
    //i_xOPN_SW :=FALSE;
    xOpen:=FALSE;
ELSIF ((rtOPN_SW.Q) AND xOPN_OK AND NOT i_xOpnLS) OR (tonOvrd.Q AND i_xOverrideMode) THEN
    q_xOPN_DO := TRUE;
END_IF
IF (xClose) AND (NOT i_xClsLS) THEN
    q_xClose_A := TRUE;
    q_xClose_B := TRUE;
    q_xClose_C := TRUE;
END_IF
IF(CloseTimer.Q) OR (i_xClsLS) THEN
    q_xClose_A := FALSE;
    q_xClose_B := FALSE;
    q_xClose_C := FALSE;
    xClose := FALSE;
    //i_xOPN_SW := FALSE;
END_IF

IF(OpenTimer.Q) AND (i_xOpnLS) THEN
    q_xOPN_DO :=  FALSE;
    i_xOPN_SW := FALSE;
    xOpen:=FALSE;
END_IF

(* Neighboring Valves Interlock bit is reset When the Vacuum event error is reset and the Shutter is opened *)
IF ((NOT i_xTrigger) OR xVeto) AND (NOT xERR_ExtFault) AND i_xOpnLS THEN
    q_xVAC_FAULT_OK := TRUE;
END_IF

(*OPN OK evaluation bit *)
xOPN_OK := (NOT xERR_ExtFault) AND (NOT i_xTrigger OR xVeto) ;

(* If Epics Command to close the Valve, check if PMPS, otherwise Keep command set to open valve *)
// is there really a PMPS requirment.



(* When the valve  is open MPS is OK*)
q_xMPS_OK := i_xOpnLS AND ((NOT i_xTrigger AND i_xPress_OK) OR xVeto)  AND NOT(i_xCLS_SW);


(* Override logic *)
(* Goal: give ability to override, but do so in a way that people won't forget it.
Solution: Override only after ten seconds of override, protect against blips,
when the valve permission goes true for more than ten seconds consistently, remove override
*)
rTrigOverrideOpen(CLK:= i_xOverrideOpen);
tonDelOK(IN:=xOPN_OK, PT:=tDelOK);
rtOK(CLK:=tonDelOK.Q);
IF rtOK.Q AND i_xOverrideOpen THEN
    i_xOverrideOpen :=FALSE;
    //if (i_xOpnLS) AND (i_xOverrideMode) THEN i_xOPN_SW := TRUE; END_IF //for seamless transition
    //Log
    fbLogger(sMsg:='Override expired', eSevr:=TcEventSeverity.Warning);
END_IF

//Override timer
tonOvrd(IN:=i_xOverrideOpen, PT:=tOvrd);


//Assign valve state
IF (i_xTrigger) THEN q_eVFS_State := E_VGC.Triggered;
ELSIF xERR_ExtFault THEN q_eVFS_State :=  E_VGC.Vac_Fault;
ELSIF NOT i_xClsLS AND tCLStimeout.Q THEN
    q_eVFS_State :=  E_VGC.Cls_Timeout;
ELSIF NOT i_xOpnLS AND tOPNtimeout.Q THEN
    q_eVFS_State :=  E_VGC.Opn_Timeout;
ELSE q_eVFS_State :=  E_VGC.At_Vac;
END_IF

(*Timers*)
CloseTimer ( IN:=xClose, PT:= TimDur, Q=>);
OpenTimer ( IN:=i_xOpnLS, PT:= OpenTimDur, Q=>);
tOPNtimeout(IN:= q_xOPN_DO, PT := tOPNTimeOutDuration);
tCLStimeout(IN:= q_xClose_A, PT := tCLSTimeOutDuration);
rtOPN_SW(CLK:= i_xOPN_SW);

(* Soft IO Mapping*)
IO();

(*Alarm reset *)
ACT_ResetAlarms();

(*FAST FAULT*)
fbFF(i_xOK := q_xMPS_OK,
    i_xReset := i_xVAC_FAULT_Reset,
    i_xAutoReset :=TRUE,
    io_fbFFHWO := io_fbFFHWO);

ACTION ACT_ResetAlarms:
//iq_stValve.xERR_DifPres R= i_xResetFault;

//iq_stValve.bErrorPresent R= i_xResetFault;

IF (NOT i_xTrigger AND i_xPress_OK AND i_xVAC_FAULT_Reset) OR xVeto THEN
    xERR_ExtFault := FALSE;
    i_xVAC_FAULT_Reset:=FALSE;
	q_xVAC_FAULT_OK := TRUE;	
END_IF


IF (i_xTrigger OR NOT i_xPress_OK) AND NOT xVeto THEN
    i_xVAC_FAULT_Reset:=FALSE;
END_IF
END_ACTION

ACTION IO:

q_xTrigger := i_xTrigger;
q_xVFS_Closed:= i_xClsLS;
q_xVFS_Open:= i_xOpnLS;
END_ACTION

END_FUNCTION_BLOCK

// ---- POUs/Functions/Valves/FB_VFS_2OO3.TcPOU
(* This function block implements basic functionality for Fast Shutter/Valves*)
(* NOTE: All 3 gauge cards with fast TTL output need to be installed in the same gauge controller*)
(* Create a separate virtual PLC for the fast shutter logic, and tie/map this task to the FAST I/O portion of the ethercat bus,
 so we can scan these I/Os faster than the rest of the vacuum I/Os.
The Fast shutter was tested with PLC task Cycle Base Time 50us with cycle time 0.050ms.*)
FUNCTION_BLOCK FB_VFS_2OO3 EXTENDS FB_Valve
VAR_INPUT
    i_xPMPS_OK : BOOL; (*External MPS interlock, Set to TRUE when no PMPS interlock is required*)
    i_xExt_OK : BOOL; (*Other External Interlock, Set to True when no external interlock is required*)
    i_sDevName : T_MaxString := 'VFS'; (*Device name for diagnostic*)
    i_xVeto_Enable : BOOL := FALSE; (*Set to TRUE if there is a Veto Valve to this VFS*)
END_VAR
VAR_IN_OUT
    io_fbFFHWO : FB_HardwareFFOutput;
END_VAR
VAR
    xOPN_OK : BOOL;         //internal variable OK to Open signal
    xERR_ExtFault : BOOL;   //internal variable External Fault signal
    xVeto : BOOL;           //internal variable Veto signal
    xTrigger : BOOL;        //internal trigger signal, output of 2oo3 logic
    xPress_OK : BOOL;       //internal signal indicating if at gauges are connected and OK
    //Fault counter triggers
    rtFault_IG1 : R_TRIG;
    rtFault_IG2 : R_TRIG;
    rtFault_IG3 : R_TRIG;
    //Reset Fault counter trigger
    rtResetFaultCounter : R_TRIG;

    //PMPS
    fbFF : FB_FastFault :=(
        i_DevName := 'VFS',
        i_Desc := 'Fault occurs when fast valve is not in open state',
        i_TypeCode := 16#1010);

    rDiffPressAllowed : REAL := 22.5;     //Torr, Default value comes from Vat Valve Manual
    rDiffPress : REAL;                    //Current pressure

    xFirstPass : BOOL := TRUE;            //Do something on first pass, after that set to FALSE

    rtOPN_SW : R_TRIG;                    //Detect rising endge on i_xOPN_SW input

    tonDelOK : TON;
    rtOK : R_TRIG;
    tonOvrd	: TON;

    tDelOK : TIME := T#60S;
    tOvrd : TIME := T#10s;
    rTrigOverrideOpen : R_TRIG;

    xClose : BOOL;
    xOpen : BOOL;
    CloseTimer : TON;
    TimDur : TIME := T#20MS;
    OpenTimer : TON;
    OpenTimDur : TIME := T#2S;

    (*Timeouts*)
    tCLSTimeOutDuration : TIME := T#0.5S;
    tOPNTimeOutDuration : TIME := T#10S;
    tOPNtimeout : TON;
    tCLStimeout : TON;


    (*IO to the valve(s)*)
    i_xOpnLS	AT%I* : BOOL; //VFS Open limit switch input
    i_xClsLS	AT%I* : BOOL; //VFS Close limit switch input
    q_xClose_A	AT%Q* : BOOL; //3x Valve Close output signals (current req.)
    q_xClose_B	AT%Q* : BOOL; //3x Valve Close output signals (current req.)
    q_xClose_C	AT%Q* : BOOL; //3x Valve Close output signals (current req.)
    q_xOPN_DO	AT%Q* : BOOL; //Valve Open output signal
    (*3x Fast trigger Inputs from CC Gauge controller.
      Make sure all tri CC gauge cards are in the same controller*)
    i_xTriggerIG1 AT%I* : BOOL; //Fast trigger input from CC gauge 1
    i_xTriggerIG2 AT%I* : BOOL; //Fast trigger input from CC gauge 2
    i_xTriggerIG3 AT%I* : BOOL; //Fast trigger input from CC gauge 3

    (*VETO Devices*)
    i_xVetoValveOpenDO AT%I* : BOOL; (*Link to VFS Interface*)
    i_xVetoValveClosed AT%I* : BOOL; (*Link to VFS Interface*)

    (*Interface with external system*)
    i_e2OO3_MODE       AT%I* : E_2OO3_MODE; (*Link to VFS Interface, 2oo3 mode selector*)
    i_ResetFaultCounter AT%I* : BOOL; (*Link to VFS Interface, FaultCounter Reset*)
    i_xPress_OK_IG1    AT%I* : BOOL; (*Link to VFS Interface, IG.xPRESS_OK, to make sure that the device is connected*)
    i_xPress_OK_IG2    AT%I* : BOOL; (*Link to VFS Interface, IG.xPRESS_OK, to make sure that the device is connected*)
    i_xPress_OK_IG3    AT%I* : BOOL; (*Link to VFS Interface, IG.xPRESS_OK, to make sure that the device is connected*)
    i_xOPN_SW          AT%I* : BOOL; (*Link to VFS Interface, external open signal e.g epics*)
    i_xCLS_SW          AT%I* : BOOL; (*Link to VFS Interface, external close signal e.g epics*)
    i_xVAC_FAULT_Reset AT%I* : BOOL; (*Link to VFS Interface Valve Vacuum OK, is set to False when there is Vacuum Fault*)
    i_xOverrideMode    AT%I* : BOOL; (*Link to VFS Interface, To be linked to global override bit. This Overrides Vacuum logic only, EPS, MPS and PMPS are still enforces*)
    i_xOverrideOpen    AT%I* : BOOL; (*Link to VFS Interface*)
    q_xTrigger         AT%Q* : BOOL; (*Link to VFS Interface*)
    q_xVFS_Open        AT%Q* : BOOL; (*Link to VFS Interface*)
    q_xVFS_Closed      AT%Q* : BOOL; (*Link to VFS Interface*)
    q_xVAC_FAULT_OK    AT%Q* : BOOL; (*Link to VFS Interface, Valve Vacuum OK, is set to False when there is Vacuum Fault*)
    q_xMPS_OK          AT%Q* : BOOL; (*Link to VFS Interface, MPS Fault OK, is set when the Valve is Open and there is no trigger*)
    q_eVFS_State       AT%Q* : E_VGC; (*Link to VFS Interface*)
    q_nFltCount_IG1    AT%Q* : UINT; (*Link to VFS Interface*)
    q_nFltCount_IG2    AT%Q* : UINT; (*Link to VFS Interface*)
    q_nFltCount_IG3    AT%Q* : UINT; (*Link to VFS Interface*)
END_VAR
VAR PERSISTENT
    nFaultCounter_IG1 : UINT;  //Fault counter for IG1
    nFaultCounter_IG2 : UINT;  //Fault counter for IG2
    nFaultCounter_IG3 : UINT;  //Fault counter for IG3
END_VAR

(*Fast Shutter/Valve Function Block*)
(*M.Ghaly Feb 2019*)
(*J. Govednik Jan 2022 Adding 2OO3 logic*)

(* Fast Shutters do not function as complete isolation valves, but are intended to rapidly limit conductance
between vacuum regions.  They should be installed in conjunction with isolation gate valves.  The conductance
of the fast shutter in the closed state may be sufficiently low as to create an isolated vacuum region.
Thus, at least a pirani gauge, that can measure a pressure down to 1x10-4 Torr, needs to be installed between
the shutter and the isolation gate valve.
In the case where a gauge is not installed, the neigboring gate Valves should not be opened unless the shutter
is Open.
*)

(*On first PLC pass, put valve into vented state, which implies a closed valve*)
IF xFirstPass THEN
    fbFF.i_DevName := i_sDevName;
    xFirstPass := FALSE;
END_IF

(*set Veto bit*)
IF (i_xVeto_Enable) THEN
    xVeto := (i_xVetoValveClosed AND NOT i_xVetoValveOpenDO);
    ELSE xVeto := FALSE;
END_IF

(*User will be able to select gauge channel or 2oo3 function*)
CASE i_e2OO3_MODE OF
    E_2OO3_MODE.MODE_2OO3:
        (*2oo3 logic*)
        //First let's verify that at least 2 gauges are connected
        xPress_OK := (i_xPress_OK_IG1 AND i_xPress_OK_IG2) OR
                      (i_xPress_OK_IG1 AND i_xPress_OK_IG3) OR
                      (i_xPress_OK_IG2 AND i_xPress_OK_IG3);

        //Each trigger input validated with Press OK bit which indicates if the gauge is connected or disconnected
        IF xPress_OK THEN
            xTrigger := ((i_xTriggerIG1 OR NOT i_xPress_OK_IG1) AND (i_xTriggerIG2 OR NOT i_xPress_OK_IG2)) OR
                        ((i_xTriggerIG1 OR NOT i_xPress_OK_IG1) AND (i_xTriggerIG3 OR NOT i_xPress_OK_IG3)) OR
                        ((i_xTriggerIG2 OR NOT i_xPress_OK_IG2) AND (i_xTriggerIG3 OR NOT i_xPress_OK_IG3));
            (*
            xTrigger := ((i_xTriggerIG1 AND i_xPress_OK_IG1) AND (i_xTriggerIG2 AND i_xPress_OK_IG2)) OR
                        ((i_xTriggerIG1 AND i_xPress_OK_IG1) AND (i_xTriggerIG3 AND i_xPress_OK_IG3)) OR
                        ((i_xTriggerIG2 AND i_xPress_OK_IG2) AND (i_xTriggerIG3 AND i_xPress_OK_IG3));
            *)
        ELSE
            xTrigger := TRUE;
        END_IF
    E_2OO3_MODE.IG1:
        xPress_OK := i_xPress_OK_IG1;
        xTrigger := i_xTriggerIG1 OR NOT i_xPress_OK_IG1;
    E_2OO3_MODE.IG2:
        xPress_OK := i_xPress_OK_IG2;
        xTrigger := i_xTriggerIG2 OR NOT i_xPress_OK_IG2;
    E_2OO3_MODE.IG3:
        xPress_OK := i_xPress_OK_IG3;
        xTrigger := i_xTriggerIG3 OR NOT i_xPress_OK_IG3;
END_CASE;

//xVeto:= i_xVeto AND (i_xVetoValveClosed AND NOT i_xVetoValveOpenDO);
(*Input Trigger to close the Fast Shutter*)
(*Neighboring Valves Should also be triggered to Close*)
//IF ((xTrigger) OR NOT (i_xPress_OK) OR NOT (i_xExt_OK))  AND NOT (xVeto) AND NOT (tonOvrd.Q AND i_xOverrideMode) THEN
IF ((xTrigger) OR NOT (i_xExt_OK))  AND NOT (xVeto) AND NOT (tonOvrd.Q AND i_xOverrideMode) THEN
    xClose := TRUE;
    xOpen := FALSE;
    q_xVAC_FAULT_OK := FALSE;
    xERR_ExtFault := TRUE;
    i_xCLS_SW := TRUE;
    q_xOPN_DO := FALSE;
    //i_xOPN_SW :=FALSE;
ELSIF (i_xCLS_SW) THEN
    xClose := TRUE;
    xOpen := FALSE;
    q_xVAC_FAULT_OK:= FALSE;
    i_xCLS_SW := TRUE;
    q_xOPN_DO := FALSE;
    //i_xOPN_SW :=FALSE;
ELSIF ((rtOPN_SW.Q) AND xOPN_OK AND NOT i_xOpnLS) OR (tonOvrd.Q AND i_xOverrideMode) THEN
    q_xOPN_DO := TRUE;
END_IF

//Hold Valve close signals to TRUE until limit swith is hit
IF (xClose) AND (NOT i_xClsLS) THEN
    q_xClose_A := TRUE;
    q_xClose_B := TRUE;
    q_xClose_C := TRUE;
END_IF

//Set Valve close signals to FALSE when close timer expires or close limit switch is closed
IF(CloseTimer.Q) OR (i_xClsLS) THEN
    q_xClose_A := FALSE;
    q_xClose_B := FALSE;
    q_xClose_C := FALSE;
    xClose := FALSE;
    //i_xOPN_SW := FALSE;
END_IF

//Set Valve open signal to FALSE when open timer expires or open limit switch is closed
IF(OpenTimer.Q) AND (i_xOpnLS) THEN
    q_xOPN_DO :=  FALSE;
    i_xOPN_SW := FALSE;
    xOpen := FALSE;
END_IF

(*Neighboring Valves Interlock bit is reset When the Vacuum event error is reset and the Shutter is opened*)
IF ((NOT xTrigger) OR xVeto) AND (NOT xERR_ExtFault) AND i_xOpnLS THEN
    q_xVAC_FAULT_OK := TRUE;
END_IF

(*OPN OK evaluation bit*)
xOPN_OK := (NOT xERR_ExtFault) AND (NOT xTrigger OR xVeto) ;

(*When the valve  is open MPS is OK*)
//q_xMPS_OK := i_xOpnLS AND ((NOT xTrigger AND i_xPress_OK) OR xVeto)  AND NOT(i_xCLS_SW);
q_xMPS_OK := i_xOpnLS AND (NOT xTrigger OR xVeto) AND NOT(i_xCLS_SW);


(*Override logic*)
(*Goal: give ability to override, but do so in a way that people won't forget it.
Solution: Override only after ten seconds of override, protect against blips,
when the valve permission goes true for more than ten seconds consistently, remove override
*)
rTrigOverrideOpen (CLK := i_xOverrideOpen); // Not used

tonDelOK (IN := xOPN_OK, PT := tDelOK);
rtOK (CLK := tonDelOK.Q);

IF rtOK.Q AND i_xOverrideOpen THEN
    i_xOverrideOpen := FALSE;
    //if (i_xOpnLS) AND (i_xOverrideMode) THEN i_xOPN_SW := TRUE; END_IF //for seamless transition
    //Log
    fbLogger(sMsg := 'Override expired', eSevr := TcEventSeverity.Warning);
END_IF

//Override timer
tonOvrd(IN := i_xOverrideOpen, PT := tOvrd);


//Assign valve state
IF (xTrigger) THEN
    q_eVFS_State := E_VGC.Triggered;
ELSIF xERR_ExtFault THEN
    q_eVFS_State :=  E_VGC.Vac_Fault;
ELSIF NOT i_xClsLS AND tCLStimeout.Q THEN
    q_eVFS_State :=  E_VGC.Cls_Timeout;
ELSIF NOT i_xOpnLS AND tOPNtimeout.Q THEN
    q_eVFS_State :=  E_VGC.Opn_Timeout;
ELSE
    q_eVFS_State :=  E_VGC.At_Vac;
END_IF

(*Timers*)
CloseTimer (IN := xClose, PT := TimDur);
OpenTimer (IN := i_xOpnLS, PT := OpenTimDur);
tOPNtimeout (IN := q_xOPN_DO, PT := tOPNTimeOutDuration);
tCLStimeout (IN := q_xClose_A, PT := tCLSTimeOutDuration);

//Detecting rising edge for i_xOPN_SW (epics command)
rtOPN_SW (CLK := i_xOPN_SW);

(*Gauge fault counters*)
rtResetFaultCounter(CLK := i_ResetFaultCounter);
IF rtResetFaultCounter.Q THEN
    nFaultCounter_IG1 := 0;
    nFaultCounter_IG2 := 0;
    nFaultCounter_IG3 := 0;
END_IF
//IG1
rtFault_IG1(CLK := i_xTriggerIG1 AND NOT xTrigger);
IF rtFault_IG1.Q THEN
    nFaultCounter_IG1 := nFaultCounter_IG1 + 1;
END_IF
//IG2
rtFault_IG2(CLK := i_xTriggerIG2 AND NOT xTrigger);
IF rtFault_IG2.Q THEN
    nFaultCounter_IG2 := nFaultCounter_IG2 + 1;
END_IF
//IG3
rtFault_IG3(CLK := i_xTriggerIG3 AND NOT xTrigger);
IF rtFault_IG3.Q THEN
    nFaultCounter_IG3 := nFaultCounter_IG3 + 1;
END_IF

(*Soft IO Mapping*)
IO();

(*Alarm reset *)
ACT_ResetAlarms();

(*FAST FAULT*)
fbFF(i_xOK := q_xMPS_OK,
    i_xReset := i_xVAC_FAULT_Reset,
    i_xAutoReset := TRUE,
    io_fbFFHWO := io_fbFFHWO);

ACTION ACT_ResetAlarms:
//iq_stValve.xERR_DifPres R= i_xResetFault;

//iq_stValve.bErrorPresent R= i_xResetFault;

IF (NOT xTrigger AND xPress_OK AND i_xVAC_FAULT_Reset) OR xVeto THEN
    xERR_ExtFault := FALSE;
    i_xVAC_FAULT_Reset := FALSE;
END_IF


IF (xTrigger OR NOT xPress_OK) AND NOT xVeto THEN
    i_xVAC_FAULT_Reset := FALSE;
END_IF
END_ACTION

ACTION IO:
q_xTrigger := xTrigger;
q_xVFS_Closed := i_xClsLS;
q_xVFS_Open := i_xOpnLS;

q_nFltCount_IG1 := nFaultCounter_IG1;
q_nFltCount_IG2 := nFaultCounter_IG2;
q_nFltCount_IG3 := nFaultCounter_IG3;
END_ACTION

END_FUNCTION_BLOCK

// ---- POUs/Functions/Valves/FB_VGC_2S.TcPOU
(* This function block implements basic functionality for turbopump isolation Valves with 2 pressure setpoints*)
(* This function block interlock is as follows:
1. The valve can be opened when the difference between the pressures on both sides is
less than the maximum differential pressure.
2. This rule persists until the pressures on both sides are lower than the vacuum-setpoints.
3. Once at-vac, the valve will close if the pressure on either side rises above the setpoint.*)
(*This function block also implements PMPS and EPS interlocks, as well as Fast MPS trigger*)
{attribute 'no_check'}
{attribute 'reflection'}
FUNCTION_BLOCK FB_VGC_2S Extends FB_Valve
VAR_IN_OUT

END_VAR
VAR_INPUT
    (*Upstream Gauge, usually ion gauge*)
    i_stUSG	:	ST_VG;
    (*Downstream Gauge, usually ion gauge*)
    i_stDSG	:	ST_VG;
    {attribute 'pytmc' := '
    pv: Dis_DPIlk
    '}
    i_xDis_DPIlk : BOOL := FALSE;  (* Set to true when calling the function to disable the differential pressure interlock *)
    i_xPMPS_OK:	BOOL	; (*Set to True To switch off the bptm and PMPS Arbiter*)
    {attribute 'pytmc' := '
    pv: EPS_OK
    '}
    i_xEPS_OK:	BOOL	:= TRUE; (*External EPS interlock, Set to TRUE when no EPS interlock is required, otherwise set to correct interlock signal*)
    i_xExt_OK: BOOL; (*Other External Interlock, Set to True when no external interlock is required. If this Valve is neigboring a Fast Shutter this should be linked to the fast shutter xVAC_FAULT_OK*)
    i_xOverrideMode : BOOL; (*To be linked to global override bit. This Overrides Vacuum logic only, EPS, MPS and PMPS are still enforces*)
    // Reset fault
    {attribute 'pytmc' := '
    pv: FF_Reset
    '}
    i_xReset: BOOL;
    i_xIsAperture:BOOL :=FALSE; // Set tp True if this is an Aperture Valve, the MPS Fault will trip only when moving.
    i_sDevName : T_MaxString :=  'VGC'; // Device name for diagnostic
    i_nTransitionRootID: UDINT; //A unique transition Root ID that is equal to or greater than 1000
END_VAR
VAR_OUTPUT
    {attribute 'pytmc' := '
    pv:
    '}
    iq_stValve : ST_VGC_2S; (* All valve data and states will be in this struct*)

    {attribute 'pytmc' := '
    pv: MPS_FAULT_OK
    field: ZNAM MPS FAULT ;
    field: ONAM MPS OK ;
    '}
    xMPS_OK:	BOOL; (*MPS Fast OK, is set when the Valve is Open*)
END_VAR
VAR_IN_OUT
    io_fbFFHWO    :    FB_HardwareFFOutput;
    fbArbiter: FB_Arbiter();
END_VAR
VAR

    // PMPS
    {attribute 'pytmc' := '
    pv: MPS_OK
    '}
    xPMPS_OK:	BOOL	; (*PMPS interlock*)
    bMoving : BOOL;
    bDone :BOOL;
    tBPTMtimeout:TON;
    bptm: BeamParameterTransitionManager;
    FFO    :    FB_FastFault :=(
        i_Desc := 'Fault occurs when the valve is not in open state',
        i_TypeCode := 16#1010);
    //g_FastFaultOutput1	:	FB_HardwareFFOutput;

    {attribute 'instance-path'}
    {attribute 'noinit'}
    sPath: STRING;

    rDiffPressAllowed	:	REAL := 22.5; // Torr, Default value comes from Vat Valve Manual
    rDiffPress : REAL;
    set : BOOL;
    reset: BOOL;

    xFirstPass	:	BOOL;
    fbFSInit		:	R_TRIG;

    tonDelOK : TON;
    rtOK	:	R_TRIG;
    tonOvrd	:	TON;
    rtOpen	:	R_TRIG;
    ftClose: F_TRIG;

    tDelOK	:	TIME := T#60S;
    tOvrd	:	TIME := T#10s;


    (* Timeouts*)
    tTimeOutDuration: TIME:= T#30S;
    tOPNtimeout: TON;
    tCLStimeout:TON;


    (*IO*)
    i_xOpnLS	AT%I*: BOOL;
    i_xClsLS	AT%I*: BOOL;
    q_xOPN_DO	AT%Q*: BOOL;

    // For logging
    eVGCPrevState : E_VGC;
END_VAR

VAR PERSISTENT
    rAT_VAC_SP	:	REAL;
    rHYST_PERC	:	REAL;
    rAT_VAC_SP_DS : REAL;
END_VAR

(* Vacuum gate valve
A. Wallace
16-10-29

A gate valve isolates vacuum volumes. Ideally it can be opened when a system is vented
to allow for faster pumping, and will close when high vacuum is lost.

The following behavior is good for valves in something like a gas attenuator.
This function block does the following:
1. The valve can be opened when the difference between the pressures on both sides is
less than the maximum differential pressure.
2. This rule persists until the pressures on both sides are lower than the vacuum-setpoint.
3. Once at-vac, the valve will close if the pressure on either side rises above the setpoint.

Alternatively, the differential pressure interlock can be disabled so the valve may only be opened
if the pressure on both sides is lower than the at-vacuum-setpoint. You want this behavior if
the valve is to be used in a UHV section.

Hysteresis is employed to ensure a smooth transition from vented/pumping down, to at-vac.

Finally, an override system is built in so you can bypass all the interlocking logic and
get back online.
*)
(* 10/1/2018 Margaret Ghaly included EPS, PMPS Checkes and MPS trigger signals*)


fbFSInit( CLK := TRUE, Q => xFirstPass);
(*IO Mapping*)
ACT_IO();

(* On first PLC pass, put valve into vented state, which implies a closed valve *)
IF xFirstPass THEN
    iq_stValve.eVGC_State := Vented;
    iq_stValve.pv_xOPN_SW := FALSE;
    FFO.i_DevName := i_sDevName;
    iq_stValve.rAT_VAC_SP_DS := 0.001;
    iq_stValve.rAT_VAC_SP := 0.001;
END_IF


///Check valve position
IF iq_stValve.i_xClsLS AND  iq_stValve.i_xOpnLS THEN
    iq_stValve.eState:=INVALID;
ELSIF NOT iq_stValve.i_xClsLS AND iq_stValve.i_xOpnLS AND iq_stValve.q_xOPN_DO THEN
    iq_stValve.eState:=OPEN;
ELSIF NOT iq_stValve.i_xClsLS AND iq_stValve.i_xOpnLS AND NOT iq_stValve.q_xOPN_DO THEN
    iq_stValve.eState:=OPEN_F;
ELSIF iq_stValve.i_xClsLS AND NOT iq_stValve.i_xOpnLS AND NOT iq_stValve.q_xOPN_DO THEN
    iq_stValve.eState:=CLOSED;
ELSIF NOT iq_stValve.i_xClsLS AND NOT iq_stValve.i_xOpnLS THEN
    iq_stValve.eState:=MOVING;
ELSE
    iq_stValve.eState:=INVALID;
END_IF

// Update hysteresis
///////////////////////////////////////////////////
IF iq_stValve.rAT_VAC_SP_LAST_DS <> iq_stValve.rAT_VAC_SP_DS OR xFirstPass THEN
    iq_stValve.rAT_VAC_SP_LAST_DS := iq_stValve.rAT_VAC_SP_DS;
    iq_stValve.rAT_VAC_HYS_DS := iq_stValve.rHYST_PERC * iq_stValve.rAT_VAC_SP_DS;
END_IF

IF iq_stValve.rAT_VAC_SP_LAST <> iq_stValve.rAT_VAC_SP OR xFirstPass THEN
    iq_stValve.rAT_VAC_SP_LAST := iq_stValve.rAT_VAC_SP;
    iq_stValve.rAT_VAC_HYS := iq_stValve.rHYST_PERC * iq_stValve.rAT_VAC_SP;
END_IF

// Setpoint one Upstream gauge
iq_stValve.rAT_VAC_HYS := LIMIT(0, iq_stValve.rAT_VAC_HYS, iq_stValve.rAT_VAC_SP);
IF iq_stValve.rAT_VAC_SP <> 0 THEN
    IF iq_stValve.rHYST_PERC <> (iq_stValve.rAT_VAC_HYS / iq_stValve.rAT_VAC_SP) THEN
        iq_stValve.rHYST_PERC := LIMIT(0, (iq_stValve.rAT_VAC_HYS / iq_stValve.rAT_VAC_SP) ,1);
    END_IF
END_IF
//setpoint two Downstream gauge
iq_stValve.rAT_VAC_HYS_DS := LIMIT(0, iq_stValve.rAT_VAC_HYS_DS, iq_stValve.rAT_VAC_SP_DS);
IF iq_stValve.rAT_VAC_SP_DS <> 0 THEN
    IF iq_stValve.rHYST_PERC <> (iq_stValve.rAT_VAC_HYS_DS / iq_stValve.rAT_VAC_SP_DS) THEN
        iq_stValve.rHYST_PERC := LIMIT(0, (iq_stValve.rAT_VAC_HYS_DS / iq_stValve.rAT_VAC_SP_DS) ,1);
    END_IF
END_IF
// Valve at vacuum check
///////////////////////////////////////////////////
    set := i_stUSG.rPRESS < iq_stValve.rAT_VAC_HYS AND i_stDSG.rPRESS < iq_stValve.rAT_VAC_HYS_DS AND i_stUSG.xPRESS_OK AND i_stDSG.xPRESS_OK;
     iq_stValve.xAT_VAC S= set;
    reset := i_stUSG.rPRESS > iq_stValve.rAT_VAC_SP OR i_stDSG.rPRESS > iq_stValve.rAT_VAC_SP_DS OR NOT i_stUSG.xPRESS_OK OR NOT i_stDSG.xPRESS_OK;
    iq_stValve.xAT_VAC R= reset;

// Differential pressure check
///////////////////////////////////////////////////
    (* Calc the differential pressure across the valve *)
    rDiffPress := ABS(i_stUSG.rPRESS - i_stDSG.rPRESS);

    (* As long as the differential pressure is less than 30mbar, the valve is allowed to open *)
    IF rDiffPress <= rDiffPressAllowed AND i_stUSG.xPRESS_OK AND i_stDSG.xPRESS_OK THEN
        iq_stValve.xDP_OK := TRUE;
    ELSE
        iq_stValve.xDP_OK	:= FALSE;
        (* If the differential pressure is exceeded, even when the valve is open,
        the state is unexpected and triggers a fault, because it suggests that something
        is wrong with the valve, or gauges or mapping or there is a major leak on one side.*)
        iq_stValve.eVGC_State := ERR_DiffPress;
        iq_stValve.xERR_DifPres := TRUE;
    END_IF

// Valve state
///////////////////////////////////////////////////
CASE iq_stValve.eVGC_State OF
    Vented: (* The Vented state is used during pump down *)
        (* Assuming the pump down went well, we are now at vacuum on both sides,
        so we move to the vacuum state, otherwise remain in the vented state *)
        IF iq_stValve.xAT_VAC AND (NOT (iq_stValve.xERR_DifPres)) AND (NOT (iq_stValve.xERR_SP)) AND (NOT (iq_stValve.xERR_ExtFault))THEN
            iq_stValve.eVGC_State := AtVacuum;
        ELSE
            iq_stValve.eVGC_State := Vented;
        END_IF

    AtVacuum:
        IF iq_stValve.xAT_VAC THEN
        (* If both pressure setpoints are made,
        then enable the differential pressure interlock, regardless of the valve state
        assuming we're using some kind of ion gauge where a pressure setpoint cannot be higher than 1E-4 T *)
        iq_stValve.eVGC_State := AtVacuum;

        ELSE

            (* If the valve is open (or in an unknown state) and either gauge is not at it's vacuum setpoint,
            we have a loss of vacuum error *)
            IF (iq_stValve.i_xOpnLS OR (NOT iq_stValve.i_xOpnLS AND NOT iq_stValve.i_xClsLS)) THEN
                iq_stValve.eVGC_State := ERR_LostVac;
                iq_stValve.xERR_SP := TRUE; //TAW changed this to the ERR_SP bool because I think that's what it was intended to be?

            (* Alternatively, if the valve is already closed and we lose pressure on one side,
            it was probably intentional venting, so we calmly move back to venting mode, and
            disable the differential pressure interlock *) //??
            ELSIF iq_stValve.i_xClsLS THEN
                iq_stValve.eVGC_State := Vented;
            END_IF

        END_IF

    ERR_DiffPress:
        IF NOT (iq_stValve.xERR_DifPres) THEN
            IF iq_stValve.xAT_VAC AND (NOT (iq_stValve.xERR_DifPres)) AND (NOT (iq_stValve.xERR_SP)) AND (NOT (iq_stValve.xERR_ExtFault))THEN
                iq_stValve.eVGC_State := AtVacuum;
            ELSE
                iq_stValve.eVGC_State := Vented;
            END_IF
        END_IF


    ERR_LostVac:
        IF NOT (iq_stValve.xERR_SP) THEN
            IF iq_stValve.xAT_VAC AND (NOT (iq_stValve.xERR_DifPres)) AND (NOT (iq_stValve.xERR_SP)) AND (NOT (iq_stValve.xERR_ExtFault))THEN
                iq_stValve.eVGC_State := AtVacuum;
            ELSE
                iq_stValve.eVGC_State := Vented;
            END_IF
        END_IF

    ERR_ExtFault:
        IF NOT (iq_stValve.xERR_ExtFault) AND (i_xExt_OK) THEN
            IF iq_stValve.xAT_VAC AND (NOT (iq_stValve.xERR_DifPres)) AND (NOT (iq_stValve.xERR_SP)) AND (NOT (iq_stValve.xERR_ExtFault))THEN
                iq_stValve.eVGC_State := AtVacuum;
            ELSE
                iq_stValve.eVGC_State := Vented;
            END_IF
        END_IF
END_CASE

IF (NOT i_xExt_OK) AND (iq_stValve.eState=OPEN)  THEN
    iq_stValve.eVGC_State := ERR_ExtFault;
    iq_stValve.xERR_ExtFault := TRUE;
END_IF

// Interlock evaluation - with bypass for DP ILK bypass
///////////////////////////////////////////////
IF i_xDis_DPIlk THEN
    iq_stValve.xOPN_OK := iq_stValve.xEXT_OK; // AND iq_stValve.xDP_OK ;
ELSE
    iq_stValve.xOPN_OK := iq_stValve.xEXT_OK AND iq_stValve.xAT_VAC;
END_IF


(* Valve operation *)

(* Override logic *)
(* Goal: give ability to override, but do so in a way that people won't forget it.
Solution: Override only after ten seconds of override, protect against blips,
when the valve permission goes true for more than ten seconds consistently, remove override
*)

tonDelOK(IN:=iq_stValve.xOPN_OK, PT:=tDelOK);
rtOK(CLK:=tonDelOK.Q);
IF rtOK.Q AND iq_stValve.pv_xOvrdOpn THEN
    iq_stValve.pv_xOvrdOpn :=FALSE;
    if (iq_stValve.eState = OPEN) AND (i_xOverrideMode) THEN iq_stValve.pv_xOPN_SW := TRUE; END_IF //for seamless transition
    //Log
    fbLogger(sMsg:='Override expired', eSevr:=TcEventSeverity.Warning);
END_IF
// Release the Force Open bit when the system override is false
IF NOT (i_xOverrideMode) THEN  iq_stValve.pv_xOvrdOpn :=FALSE; END_IF
//Override timer
tonOvrd(IN:=iq_stValve.pv_xOvrdOpn, PT:=tOvrd);


(* Valve operation *)
(* Here's where we evaluate sw actions and operate the valve *)
(* Valve operation *)

ftClose(CLK:= iq_stValve.pv_xOPN_SW);
rtOpen(CLK:= iq_stValve.pv_xOPN_SW);


(*PMPS*)
IF NOT(i_xPMPS_OK) THEN
    ACT_PMPS();
END_IF
(*when interlock is lost the Valve closes regardless of the status of the PMPS and EPS*)
xPMPS_OK := i_xPMPS_OK OR (bptm.q_xTransitionAuthorized OR tBPTMtimeout.Q);
IF NOT (iq_stValve.xOPN_OK) THEN
    iq_stValve.pv_xOPN_SW:= FALSE; // Reset switch after inlk is lost
    iq_stValve.q_xOPN_DO := (iq_stValve.pv_xOPN_SW  AND iq_stValve.xOPN_OK) OR (tonOvrd.Q AND i_xOverrideMode);
ELSIF xPMPS_OK THEN
    iq_stValve.q_xOPN_DO := (iq_stValve.pv_xOPN_SW  AND iq_stValve.xOPN_OK) OR (tonOvrd.Q AND i_xOverrideMode);
//ELSIF NOT (i_xPMPS_OK) THEN
    // Only override mode
    //iq_stValve.q_xOPN_DO := (tonOvrd.Q AND i_xOverrideMode);
END_IF


(*MPS Fault setting*)
If (i_xIsAperture ) THEN
    (* When the valve  is open or in Closed position MPS is OK, Fault while moving*)
    xMPS_OK := (i_xOpnLS  AND q_xOPN_DO) XOR (i_xClsLS  AND NOT q_xOPN_DO);
ELSE
    (* When the valve  is open MPS is OK*)
    xMPS_OK := i_xOpnLS AND NOT i_xClsLS AND q_xOPN_DO;
END_IF


///Check valve moving postion timout
IF NOT iq_stValve.i_xClsLS AND tCLStimeout.Q THEN
    iq_stValve.bErrorPresent := TRUE;
    iq_stValve.sErrorMessage := 'Close Timeout';
ELSIF NOT iq_stValve.i_xOpnLS AND tOPNtimeout.Q THEN
    iq_stValve.bErrorPresent := TRUE;
    iq_stValve.sErrorMessage := 'Open Timeout';
END_IF
IF (iq_stValve.eState=INVALID) THEN
    iq_stValve.bErrorPresent := TRUE;
    iq_stValve.sErrorMessage := CONCAT(sPath,'Invalid Valve Position');
END_IF


(*Timers*)
tOPNtimeout(IN:= iq_stValve.q_xOPN_DO, PT := tTimeOutDuration );
tCLStimeout(IN:= NOT iq_stValve.q_xOPN_DO, PT := tTimeOutDuration);


// Alarm reset
//////////////////////////////////////
ACT_ResetAlarms();

(*IO Mapping*)
ACT_IO();

// Log States and triggers
ACT_Logger();

(*Load or save the persistent variables*)
ACT_Persistent();

(*FAST FAULT*)
FFO(i_xOK := xMPS_OK,
    i_xReset := i_xReset,
    i_xAutoReset :=TRUE,
    i_DevName := i_sDevName,
    io_fbFFHWO := io_fbFFHWO);

ACTION ACT_IO:
(*inputs*)
iq_stValve.i_xOpnLS := 	i_xOpnLS;
iq_stValve.i_xClsLS:=	i_xClsLS;
iq_stValve.xEXT_OK := i_xEXT_OK;
iq_stValve.xOverrideMode := i_xOverrideMode;
(*outputs*)
q_xOPN_DO:= iq_stValve.q_xOPN_DO;

(*ILK Devices*)
iq_stValve.sIlkUSDeviceName := This^.i_stUSG.sPath;
iq_stValve.sIlkDSDeviceName := This^.i_stDSG.sPath;
END_ACTION

ACTION ACT_Logger:
// ILK logger

IF NOT (iq_stValve.xOPN_OK) AND (ePrevState = OPEN) AND NOT (TonOvrd.Q) THEN
         fbLogger(sMsg:='Lost interlock ok bit while valve was open.', eSevr:=TcEventSeverity.Critical);
END_IF


//Positiong STATE Logger
IF ePrevState <> iq_stValve.eState THEN
      CASE iq_stValve.eState OF
        INVALID:
            fbLogger(sMsg:='Valve invalid position.', eSevr:=TcEventSeverity.Critical);
          MOVING:
            fbLogger(sMsg:='Valve moving', eSevr:=TcEventSeverity.Warning);
        OPEN:
            fbLogger(sMsg:='Valve Open.', eSevr:=TcEventSeverity.Info);
        OPEN_F:
            fbLogger(sMsg:='Valve Open.', eSevr:=TcEventSeverity.Info);
        CLOSED:
            fbLogger(sMsg:='Valve closed.', eSevr:=TcEventSeverity.Info);
      END_CASE
      ePrevState := iq_stValve.eState;
  END_IF

 //Pressure STATE Logger
IF eVGCPrevState <> iq_stValve.eVGC_State THEN
      CASE iq_stValve.eVGC_State OF
        Vented:
             fbLogger(sMsg:='Vented', eSevr:=TcEventSeverity.Info);
          AtVacuum:
             fbLogger(sMsg:='Vacuum setpoint satisfied', eSevr:=TcEventSeverity.Info);
        ERR_DiffPress:
             fbLogger(sMsg:='Potential accidental vent.', eSevr:=TcEventSeverity.Critical);
        ERR_LostVac:
            fbLogger(sMsg:='Unexpected loss of vacuum while valve was open or moving.', eSevr:=TcEventSeverity.Critical);
        ERR_ExtFault:
             fbLogger(sMsg:='Lost external interlock while valve was open.', eSevr:=TcEventSeverity.Critical);
      END_CASE
      eVGCPrevState := iq_stValve.eVGC_State;
  END_IF



// Log valve timeouts
tErrorPresent(CLK:=iq_stValve.bErrorPresent);
IF tErrorPresent.Q THEN fbLogger(sMsg:=iq_stValve.sErrorMessage, eSevr:=TcEventSeverity.Warning); END_IF

// Log valve open
tAction(CLK:= iq_stValve.q_xOPN_DO);
IF tAction.Q THEN fbLogger(sMsg:='Valve commanded open', eSevr:=TcEventSeverity.Info); END_IF

// Log override mode enabled
tOverrideActivated(CLK:= (tonOvrd.Q AND i_xOverrideMode));
IF tOverrideActivated.Q THEN fbLogger(sMsg:='Valve override mode activated', eSevr:=TcEventSeverity.Warning); END_IF
END_ACTION

ACTION ACT_Persistent:
(*On first PLC pass, load the persistent value into the structrue variable*)
IF (SUPER^.bRestorePersistentData) THEN
    SUPER^.bRestorePersistentData	:= FALSE;
    IF (rAT_VAC_SP <> 0) THEN
        iq_stValve.rAT_VAC_SP := rAT_VAC_SP;
    END_IF;
    IF (rHYST_PERC <> 0) THEN
            iq_stValve.rHYST_PERC := rHYST_PERC;
    END_IF;
    IF (rAT_VAC_SP_DS <> 0) THEN
        iq_stValve.rAT_VAC_SP_DS := rAT_VAC_SP_DS;
    END_IF;
END_IF
(*Check if a new value has been written in the structure variable copy it to the persistent variable*)
IF NOT (iq_stValve.rAT_VAC_SP = rAT_VAC_SP) THEN
    rAT_VAC_SP := iq_stValve.rAT_VAC_SP;
END_IF;

IF NOT (iq_stValve.rAT_VAC_HYS = rHYST_PERC) THEN
    rHYST_PERC := iq_stValve.rAT_VAC_HYS;
END_IF;

IF NOT (iq_stValve.rAT_VAC_SP_DS = rAT_VAC_SP_DS) THEN
    rAT_VAC_SP_DS := iq_stValve.rAT_VAC_SP_DS;
END_IF;
END_ACTION

ACTION ACT_PMPS:
bMoving := (iq_stValve.pv_xOPN_SW AND iq_stValve.i_xClsLS) XOR (NOT iq_stValve.pv_xOPN_SW AND i_xOpnLS);
bDone := (iq_stValve.pv_xOPN_SW AND iq_stValve.i_xOpnLS) XOR (NOT iq_stValve.pv_xOPN_SW AND i_xClsLS);
If (i_xIsAperture ) OR (iq_stValve.pv_xOPN_SW )THEN
    bptm.i_stRequestedAssertion := PMPS_GVL.cstFullBeam;
ELSE  bptm.i_stRequestedAssertion := PMPS_GVL.cst0RateBeam;
END_IF
bptm(fbArbiter:=fbArbiter,
     i_sDeviceName:=i_sDevName,
     i_TransitionAssertionID:=i_nTransitionRootID+2,
     i_stTransitionAssertion:=PMPS_GVL.cst0RateBeam,
     i_nRequestedAssertionID:=i_nTransitionRootID+ BOOL_TO_UDINT( iq_stValve.pv_xOPN_SW),
     i_stRequestedAssertion:=,
     i_xMoving:=bMoving,
     i_xDoneMoving:= bDone,
     stCurrentBeamParameters:=PMPS_GVL.stCurrentBeamParameters,
     q_xTransitionAuthorized=>);
// Timeout
tBPTMtimeout(IN:= bMoving AND NOT bptm.q_xTransitionAuthorized , PT:=T#1S);
//xPMPS_OK := bptm.q_xTransitionAuthorized OR tBPTMtimeout.Q;

//Timeout and clear request
IF (tBPTMtimeout.Q) THEN
    fbArbiter.RemoveRequest(bptm.i_TransitionAssertionID);
    fbArbiter.RemoveRequest(bptm.i_nRequestedAssertionID);
END_IF
END_ACTION

ACTION ACT_ResetAlarms:
iq_stValve.xERR_DifPres R= iq_stValve.pv_xAlmRst;
iq_stValve.xERR_SP R= iq_stValve.pv_xAlmRst;
iq_stValve.bErrorPresent R= iq_stValve.pv_xAlmRst;
iq_stValve.xERR_ExtFault R= iq_stValve.pv_xAlmRst;

IF ( iq_stValve.pv_xAlmRst) THEN
    iq_stValve.sErrorMessage :='';
     iq_stValve.pv_xAlmRst := FALSE;
END_IF
END_ACTION

METHOD PUBLIC M_IsClosed : BOOL
VAR_INPUT
END_VAR
M_IsClosed := (This^.iq_stValve.eState = E_ValvePositionState.CLOSED);
END_METHOD

METHOD PUBLIC M_IsOpen : BOOL
VAR_INPUT
END_VAR
M_IsOpen := (This^.iq_stValve.eState = E_ValvePositionState.OPEN);
END_METHOD

// Use this Methode to Open or close the valve by setting the OPN_SW to the input value.
METHOD PUBLIC M_Set_OPN_SW : BOOL
VAR_INPUT
        value:BOOL;
END_VAR
This^.iq_stValve.pv_xOPN_SW := value;
END_METHOD

END_FUNCTION_BLOCK

// ---- POUs/Functions/Valves/FB_VRC_DA.TcPOU
(* This Function Block Implements Basic Functionality for dual acting valves. EPs is implemented so that there is interlock Open and Interlock close,
This function block is interloked by an input . This is so developers can interface with custom
interlocking logic outside this function block.*)
(* Note Interlock Logic is External *)
{attribute 'no_check'}
FUNCTION_BLOCK FB_VRC_DA EXTENDS FB_Valve
VAR_IN_OUT

END_VAR
VAR_INPUT
    i_OPN_OK : BOOL; //Connect to EPS Interlock logic condition, Set to True if the valve is not interlocked
    i_CLS_OK : BOOL; //Connect to EPS Interlock logic condition, Set to True if the valve is not interlocked
    ibCntrlHold:BOOL; (* Control Signal must retain its value, False in case of pulse control*)

    i_xOverrideMode : BOOL; (*To be linked to global override bit. This Overrides Vacuum logic only, EPS, MPS and PMPS are still enforces*)
END_VAR
VAR_OUTPUT
    {attribute 'pytmc' := '
    pv:
    '}
    iq_stValve : ST_VRC_NO;
END_VAR
VAR
    {attribute 'instance-path'}
    {attribute 'noinit'}
    sPath: STRING;
    xFirstPass	:	BOOL;
    fbFSInit		:	R_TRIG;
    tonOvrd	:	TON;
    tonDelOK : TON;
    rtOK	:	R_TRIG;
    tOvrd	:	TIME := T#10s;
    (* Timeouts*)
    tTimeOutDuration: TIME:= T#30S;
    tOPNtimeout: TON;
    tCLStimeout:TON;
    (*Limit switch latch timer*)
    tLimitSwitchLatchDuration: TIME:=T#1S;
    tOPNLimitSwitch:TON;
    tCLSLimitSwitch:TON;
    tAction2 : R_TRIG;
    (*IO*)
    i_xOpnLS	AT%I*: BOOL;
    i_xClsLS	AT%I*: BOOL;
    q_xOPN_DO	AT%Q*: BOOL;
    q_xCLS_DO	AT%Q*: BOOL;

END_VAR


(* On first PLC pass, put valve into vented state, which implies a closed valve *)
fbFSInit( CLK := TRUE, Q => xFirstPass);
IF xFirstPass THEN
    iq_stValve.eVGC_State := Vented;
    iq_stValve.pv_xOPN_SW := FALSE;
    iq_stValve.pv_xCLS_SW := FALSE;
    ePrevState := INVALID;
END_IF


///Check valve position
IF iq_stValve.i_xClsLS AND  iq_stValve.i_xOpnLS THEN
    iq_stValve.eState:=INVALID;
ELSIF NOT iq_stValve.i_xClsLS AND iq_stValve.i_xOpnLS THEN
    iq_stValve.eState:=OPEN;
ELSIF iq_stValve.i_xClsLS AND NOT iq_stValve.i_xOpnLS THEN
    iq_stValve.eState:=CLOSED;
ELSIF NOT iq_stValve.i_xClsLS AND NOT iq_stValve.i_xOpnLS THEN
    iq_stValve.eState:=MOVING;
ELSE
    iq_stValve.eState:=INVALID;
END_IF



(* Can't have both open and close True at the same time. Reset both*)
If (iq_stValve.pv_xOPN_SW) AND (iq_stValve.pv_xCLS_SW) THEN
    iq_stValve.pv_xOPN_SW := FALSE;
    iq_stValve.pv_xCLS_SW := FALSE;
END_IF

(* Override logic *)
(* Goal: give ability to override, but do so in a way that people won't forget it.
Solution: Override only after ten seconds of override, protect against blips,
when the valve permission goes true for more than ten seconds consistently, remove override
*)


// Release the Force Open bit when the system override is false
IF NOT(i_xOverrideMode) THEN
    iq_stValve.pv_xOvrdOpn :=FALSE;
    iq_stValve.pv_xOvrdCls := FALSE;
END_IF
//Override timer
tonOvrd(IN:=(iq_stValve.pv_xOvrdOpn OR iq_stValve.pv_xOvrdCls), PT:=tOvrd);

(* Here's where the valve Actuates *)
(*Evaluate EPS interlocks and the override*)
iq_stValve.q_xCLS_DO  := (i_CLS_OK AND iq_stValve.pv_xCLS_SW AND NOT iq_stValve.pv_xOPN_SW) OR (tonOvrd.Q AND iq_stValve.pv_xOvrdCls AND i_xOverrideMode);
iq_stValve.q_xOPN_DO  := (i_OPN_OK AND iq_stValve.pv_xOPN_SW AND NOT iq_stValve.pv_xCLS_SW) OR (tonOvrd.Q AND iq_stValve.pv_xOvrdOpn AND i_xOverrideMode) ;

